(**********************************************Mesure debit ByPass*)
(*******Convertion de la pression en débit**********)
Calcul_5 := EXPT(Tab_MES_Sonde_Press_ByPass.R_MesCor,2);
Calcul_6 := EXPT(Tab_MES_Sonde_Press_ByPass.R_MesCor,1);
MES_Debit_ByPass_m3h :=  (0.0035 * Calcul_5) + (0.8986 * Calcul_6) + 10.289;

(*******Mise à zéro de la mesure en cas d'arrête*********)
TON_P1(IN:= (TON_F6.Q OR NOT Option_Mot_ByPass), PT:= T#2s);
IF (TON_P1.Q)
	THEN
	MES_Debit_ByPass_m3h := 0.0;
	ELSE
	MES_Debit_ByPass_m3h := MES_Debit_ByPass_m3h;
END_IF;

(**********************************************Mesure debit extraction et soufflage en Vol/h*)
Filtre_V1_Extraction(Mesure:= Tab_MES_Sonde_Gros_Debit_Extraction.R_MesCor, Temps_Echantillonage:= T#2s);
Filtre_V1_Soufflage(Mesure:= Tab_MES_Sonde_Gros_Debit_Soufflage.R_MesCor, Temps_Echantillonage:= T#2s);
Filtre_V1_BasDebit(Mesure:= MES_Petit_Debit_m3h_Extraction, Temps_Echantillonage:= T#1s);
Filtre_V1_ByPass(Mesure:= MES_Debit_ByPass_m3h, Temps_Echantillonage:= T#1s);

IF (Enable_PID_Bas_Deb_Ext)
	THEN
	MES_Debit_Volh_Soufflage 		:= MES_Petit_Debit_m3h_Extraction / MAX(1,Volume_Cabine);
ELSE
	MES_Debit_Volh_Soufflage			:= Filtre_V1_Soufflage.Mesure_Echantillonner / MAX(1,Volume_Cabine);
END_IF;
MES_Debit_Volh_Extraction 		:= Filtre_V1_Extraction.Mesure_Echantillonner / MAX(1,Volume_Cabine);
MES_Petit_Debit_Volh_Extraction 	:= MES_Petit_Debit_m3h_Extraction / MAX(1,Volume_Cabine);
MES_Debit_ByPass_Volh 			:= Filtre_V1_ByPass.Mesure_Echantillonner / MAX(1,Volume_Cabine);

(**********************************************Mesure de la temperature d'ambiance en °F*)
MES_Sonde_Temp_Amb_F := LIMIT(0.0, ((Tab_MES_Sonde_Temp_Amb.R_MesCor * 1.8) + 32), 100.0);

(**********************************************Mesure de la temperature de l'eau mitige de l'arrivée d'eau en °C et °F*)
IF(Option_Sonde_Temp_EauMitig) (*Option gestion régulation température eau mitigée*)
	THEN
	MES_Temp_Eau_Mitige_Cabine := Tab_MES_Sonde_Temp_Eau_Mitig.R_MesCor;
	MES_Temp_Eau_Mitige_Cabine_F := (MES_Temp_Eau_Mitige_Cabine * 1.8) + 32;
	ELSE
	MES_Temp_Eau_Mitige_Cabine := 0.0;
	MES_Temp_Eau_Mitige_Cabine_F := 0.0;
END_IF;

(**********************************************Mesure de la temperature de l'eau mitige de l'arrivée d'eau en °C et °F*)
IF(Option_Vanne_Thermo_General) (*Option vanne thermostatique présente pour toute les cabines*)
	THEN
	MES_Temp_Eau_Mitige_General_F := INT_TO_REAL(Temp_Eau_Mitige) / 10.0;
	MES_Temp_Eau_Mitige_General := LIMIT(0.0, ((MES_Temp_Eau_Mitige_General_F - 32.0) / 1.8), 100.0);
	ELSE
	MES_Temp_Eau_Mitige_General_F := 0.0;
	//MES_Temp_Eau_Mitige_General := 0.0;
END_IF;

(**********************************************Mesure sonde de pression de soufflage general*)
IF(Option_Press_SoufExt_General) (*Gestion des options*)
	THEN	E_Sonde_press_Souf := E_Sonde_press_Souf;
	ELSE	E_Sonde_press_Souf := 0;
END_IF;

(*Objet sonde*)
Objet_Sonde_V1_Press_Souf(
	Mesure_EAN:= INT_TO_REAL(E_Sonde_press_Souf),
	Enable_Alarme:= TRUE,
	Status_DEF_EAN:= FALSE,
	Tempo_AL:= T#60s,
	Hyst_AL:= 1.0,
	EAN_MIN:= 0.0,
	EAN_MAX:= 32767.0,
	MES_MIN:= 0.0,
	MES_MAX:= 500.0,
	Filtre_Actif:= TRUE,
	Temps_Echantillonage:= T#500ms,
	Tab_Sonde:= Tab_Mes_Sonde_Pression_Souf);
Tab_Mes_Sonde_Pression_Souf.R_MesCor := Tab_Mes_Sonde_Pression_Souf.R_MesCor;

(**********************************************Mesure sonde de pression d'extraction general*)
IF(Option_Press_SoufExt_General) (*Gestion des options*)
	THEN	E_Sonde_press_Ext := E_Sonde_press_Ext;
	ELSE	E_Sonde_press_Ext := 0;
END_IF;

(*Objet sonde*)
Objet_Sonde_V1_Press_Ext(
	Mesure_EAN:= INT_TO_REAL(E_Sonde_press_Ext),
	Enable_Alarme:= TRUE,
	Status_DEF_EAN:= FALSE,
	Tempo_AL:= T#60s,
	Hyst_AL:= 1.0,
	EAN_MIN:= 0.0,
	EAN_MAX:= 32767.0,
	MES_MIN:= 0.0,
	MES_MAX:= 500.0,
	Filtre_Actif:= TRUE,
	Temps_Echantillonage:= T#500ms,
	Tab_Sonde:= Tab_Mes_Sonde_Pression_Ext);
Tab_Mes_Sonde_Pression_Ext.R_MesCor := Tab_Mes_Sonde_Pression_Ext.R_MesCor;

(*********************************************Mesure sonde de température batterie eau glacée*)
IF(Option_Temp_Batterie_EG) (*Gestion des options*)
	THEN	E_Sonde_Temp_Batt_EG := E_Sonde_Temp_Batt_EG;
	ELSE	E_Sonde_Temp_Batt_EG := 0;
END_IF;

(*Objet sonde*)
Objet_Sonde_Temp_Batt_EG(
	Mesure_EAN:= INT_TO_REAL(E_Sonde_Temp_Batt_EG),
	Enable_Alarme:= FALSE,
	Status_DEF_EAN:= FALSE,
	Tempo_AL:= T#60s,
	Hyst_AL:= 1.0,
	EAN_MIN:= 0.0,
	EAN_MAX:= 32767.0,
	MES_MIN:= -15.0,
	MES_MAX:= 35.0,
	Filtre_Actif:= FALSE,
	Temps_Echantillonage:= T#1s,
	Tab_Sonde:= Tab_Mes_Sonde_Temp_BatEG);
Tab_Mes_Sonde_Temp_BatEG.R_MesCor := Tab_Mes_Sonde_Temp_BatEG.R_MesCor;

(*********************************************Mesure sonde de température au soufflage*)
IF(TRUE) (*Gestion des options*)
	THEN	E_Sonde_Temp_Souf := E_Sonde_Temp_Souf;
	ELSE	E_Sonde_Temp_Souf := 0;
END_IF;

(*Objet sonde*)
Objet_Sonde_Temp_Souf(
	Mesure_EAN:= INT_TO_REAL(E_Sonde_Temp_Souf),
	Enable_Alarme:= TRUE,
	Status_DEF_EAN:= Defaut_Sonde_Temp_Souf,
	Tempo_AL:= T#5S,
	Hyst_AL:= 1.0,
	EAN_MIN:= 0.0,
	EAN_MAX:= 32767.0,
	MES_MIN:= -20.0,
	MES_MAX:= 80.0,
	Filtre_Actif:= FALSE,
	Temps_Echantillonage:= T#1s,
	Tab_Sonde:= Tab_Mes_Sonde_Temp_Souf);
Tab_Mes_Sonde_Temp_Souf.R_MesCor := Tab_Mes_Sonde_Temp_Souf.R_MesCor;

END_PROGRAM

// ---- POUs/Block/Objets/Objet_Sonde_V1.TcPOU
FUNCTION_BLOCK Objet_Sonde_V1
VAR_INPUT
	Mesure_EAN: REAL;
	Enable_Alarme: BOOL;
	Status_DEF_EAN: BOOL;
	Tempo_AL: TIME;
	Hyst_AL: REAL;
	EAN_MIN: REAL;
	EAN_MAX: REAL;
	MES_MIN: REAL;
	MES_MAX: REAL;
	Filtre_Actif: BOOL;
	Temps_Echantillonage: TIME;
END_VAR

VAR
	TON_AL_S: TON;
	TON_AL_B: TON;
	TON_AL_H: TON;
	TON_1: TON;
	TON_2: TON;
	TP_1: TP;
	TP_2: TP;
	R_TRIG_1: R_TRIG;
	R_TRIG_2: R_TRIG;
	val_a: REAL;
	val_b: REAL;
	val_y: REAL;
	val_x: REAL;
	val_1: REAL;
	val_2: REAL;
	Diff_Mesure: REAL;
	Mesure_Echantillonner: REAL;
	Incremment_Mesure: REAL;
	Incremment_Temps: TIME;
	DINT_Temps_Echantillonage: DINT;
	DINT_Incremment_Temps: DINT;
END_VAR
VAR_IN_OUT
	Tab_Sonde :Objet_Sonde;
END_VAR

(* Gestion mesure **************************************************************)
(* Mise à l'échelle température *)
val_1 := MES_MAX - MES_MIN;
val_2 := EAN_MAX - EAN_MIN;
val_x := Mesure_EAN;
val_a := val_1 / MAX(0.1,val_2);
val_b := MES_MAX - (val_a * EAN_MAX);
val_y := (val_a * val_x) + val_b;
Tab_Sonde.R_MesBrut := LIMIT(MES_MIN,val_y,MES_MAX);

(* Gestion filtrage mesure *)
(* Fonction échantillonnage ***************)
TON_1(IN := NOT(TP_1.Q), PT := Temps_Echantillonage);
TP_1(IN := TON_1.Q , PT := T#500ms);

(* Calcule de l'éccart entre la mesure et mesure T-1 ***************) 
R_TRIG_1(CLK := TP_1.Q);
IF R_TRIG_1.Q
	THEN
		Diff_Mesure := Tab_Sonde.R_MesBrut - Mesure_Echantillonner;
END_IF;

(* Détermination de l'incremment ***************)
Incremment_Mesure := Diff_Mesure / 10.0;

(* Détermination du temps entre chaque incremmentation ***************) 
DINT_Temps_Echantillonage := TIME_TO_DINT(Temps_Echantillonage) / 1000;
DINT_Incremment_Temps := DINT_Temps_Echantillonage;
Incremment_Temps := DINT_TO_TIME(DINT_Incremment_Temps * 1000);

(* Echantillonage de la mesure ***************) 
(* Temporisation d'incrementation *)
TON_2(IN := NOT(TP_2.Q), PT := Incremment_Temps);
TP_2(IN := TON_2.Q , PT := T#100ms);

R_TRIG_2(CLK := TP_2.Q);
IF R_TRIG_2.Q
	THEN
		Mesure_Echantillonner := Mesure_Echantillonner + Incremment_Mesure;
END_IF;

(* Calcule mesure température corrigé *)
IF Filtre_Actif
	THEN
		Tab_Sonde.R_MesCor := Mesure_Echantillonner + Tab_Sonde.W_Offset;
	ELSE
		Tab_Sonde.R_MesCor := Tab_Sonde.R_MesBrut + Tab_Sonde.W_Offset;
END_IF;

(* Gestion alarmes *************************************************************)
(* Alarme status température *)
TON_AL_S(IN := Status_DEF_EAN, PT := Tempo_AL);
Tab_Sonde.Mot_Lecture.0 := TON_AL_S.Q;

(* Alarme température basse *)
TON_AL_B(IN := (Tab_Sonde.R_MesCor < Tab_Sonde.W_SeuilAlarmeBasse) AND Enable_Alarme, PT := Tempo_AL);
IF TON_AL_B.Q
	THEN
		Tab_Sonde.Mot_Lecture.2 := TRUE;
END_IF;
IF ((Tab_Sonde.R_MesCor - Hyst_AL) >= Tab_Sonde.W_SeuilAlarmeBasse OR NOT (Enable_Alarme))
	THEN
		Tab_Sonde.Mot_Lecture.2 := FALSE;
END_IF;

(* Alarme température haute *)
TON_AL_H(IN := (Tab_Sonde.R_MesCor > Tab_Sonde.W_SeuilAlarmeHaute) AND Enable_Alarme, PT := Tempo_AL);
IF TON_AL_H.Q
	THEN
		Tab_Sonde.Mot_Lecture.1 := TRUE;
END_IF;
IF ((Tab_Sonde.R_MesCor + Hyst_AL) <= Tab_Sonde.W_SeuilAlarmeHaute OR NOT (Enable_Alarme))
	THEN
		Tab_Sonde.Mot_Lecture.1 := FALSE;
END_IF;

END_FUNCTION_BLOCK

// ---- POUs/Block/Autres/Filtre_V1.TcPOU
FUNCTION_BLOCK Filtre_V1
VAR_INPUT
	Mesure: REAL;
	Temps_Echantillonage: TIME;
END_VAR
VAR_OUTPUT
	Mesure_Echantillonner: REAL;
END_VAR
VAR
	Diff_Mesure: REAL;
	Incremment_Mesure: REAL;
	Incremment_Temps: TIME;
	DINT_Temps_Echantillonage: DINT;
	DINT_Incremment_Temps: DINT;
	TON_1: TON;
	TP_1: TP;
	R_TRIG_1: R_TRIG;
	TON_2: TON;
	TP_2: TP;
	R_TRIG_2: R_TRIG;
	Temps_Ecoule: TIME;
	Temps_Incremment: TIME;
END_VAR

(* Fonction échantillonnage ***************)
TON_1(IN := NOT(TP_1.Q), PT := Temps_Echantillonage);
Temps_Ecoule := TON_1.ET;
TP_1(IN := TON_1.Q , PT := T#500ms);

(* Calcule de l'éccart entre la mesure et mesure T-1 ***************)
R_TRIG_1(CLK := TP_1.Q);
IF R_TRIG_1.Q
	THEN
		Diff_Mesure := Mesure - Mesure_Echantillonner;
END_IF;

(* Détermination de l'incremment ***************) 
Incremment_Mesure := Diff_Mesure / 10.0;

(* Détermination du temps entre chaque incremmentation ***************) 
DINT_Temps_Echantillonage := TIME_TO_DINT(Temps_Echantillonage) / 1000;
DINT_Incremment_Temps := DINT_Temps_Echantillonage;
Incremment_Temps := DINT_TO_TIME(DINT_Incremment_Temps * 1000);

(* Echantillonage de la mesure ***************) 
(* Temporisation d'incrementation *)
TON_2(IN := NOT(TP_2.Q), PT := Incremment_Temps);
Temps_Incremment := TON_2.ET;
TP_2(IN := TON_2.Q , PT := T#100ms);

R_TRIG_2(CLK := TP_2.Q);
IF R_TRIG_2.Q
	THEN
		Mesure_Echantillonner := Mesure_Echantillonner + Incremment_Mesure;
END_IF;

END_FUNCTION_BLOCK

// ---- POUs/Block/Autres/SCL.TcPOU
FUNCTION_BLOCK SCL
VAR_INPUT
	IN_INT: INT;
	LIM_MIN_IN_REAL: REAL;
	LIM_MAX_IN_REAL: REAL;
	LIM_MIN_OUT_REAL: REAL;
	LIM_MAX_OUT_REAL: REAL;
END_VAR
VAR_OUTPUT
	OUT_REAL: REAL;
	OUT_INT: INT;
END_VAR
VAR
	val_final: REAL;
	TON_1: TON;
	SCL_OUT: REAL;
	TON_2: TON;
	val_b: REAL;
	val_a: REAL;
	val_y: REAL;
	val_x: REAL;
	LIM_MAX_IN: REAL;
	LIM_MAX_OUT: REAL;
	SCL_IN: REAL;
END_VAR

(* Sécurité anti division / 0 *)

TON_1(IN := TRUE, PT := t#1s);
LIM_MAX_IN := SEL(TON_1.Q, 1.0, LIM_MAX_IN_REAL);

IF ((LIM_MAX_IN - LIM_MIN_IN_REAL) = 0.0)
	THEN
		SCL_IN := 1.0;
	ELSE
		SCL_IN := LIM_MAX_IN - LIM_MIN_IN_REAL;
END_IF;

TON_2(IN := TRUE, PT := t#1s);
LIM_MAX_OUT := SEL(TON_2.Q, 1.0, LIM_MAX_OUT_REAL);

IF ((LIM_MAX_OUT - LIM_MIN_OUT_REAL) = 0.0)
	THEN
		SCL_OUT := 1.0;
	ELSE
		SCL_OUT := LIM_MAX_OUT - LIM_MIN_OUT_REAL;
END_IF;

(* Mise à l'échelle *)

val_x := INT_TO_REAL(IN_INT);

val_b := LIM_MAX_OUT_REAL - (val_a * LIM_MAX_IN_REAL);

val_a := (SCL_OUT) / MAX(0.1,(SCL_IN));

val_y := (val_a * val_x) + val_b;


(* Traitement final *)

val_final := val_y;
OUT_REAL := LIMIT(0.0, val_final, LIM_MAX_OUT_REAL);
OUT_INT := REAL_TO_INT(OUT_REAL);

END_FUNCTION_BLOCK

// ---- POUs/c_Gestion_Defaut.TcPOU
PROGRAM c_Gestion_Defaut
VAR
(*Gestion du defaut débordement du bac à douche*)
	TON_1: TON;
	RS_Def_Debord_Douche: RS;
(*Gestion du defaut débordement du lavabo*)
	TON_2: TON;
	RS_Def_Debord_Lavabo: RS;
(*Alarme Discordance débit d'eau de douche*)
	TON_3: TON;
	RS_Deb_Eau_Douche: RS;
(*Alarme Discordance débit d'eau du lavabo*)
	TON_4: TON;
	RS_Deb_Eau_Lavabo: RS;
(*Gestion du défaut de discordance de la prise de courant*)
	TON_5: TON;
	RS_Discord_Prise: RS;
(*Gestion du défaut de discordance alimentation de la prise (si contacteur forcé manuellement)*)
	TON_6: TON;
	RS_Forcage_Prise: RS;
(*Coupure prise en cas d'ouverture de la porte lors d'une recette en cours*)
	Mode_Prise_En_Cours: BOOL;
	RS_Porte_Ouv_Cycle: RS;
(*Gestion du defaut pompe de relevage*)
	TON_7: TON;
(*Gestion du defaut ouverture de la porte trop longue*)
	TON_8: TON;
(*Gestion des défauts de communication du module dalcnet*)
	TON_ComDalcnet :TON;
	RS_Def_Com_Dalcnet: RS;
(*Gestion des défauts de communication de la vanne thermostatique otpion sur chaque cabine*)
	TON_Thermo :TON;
	RS_Def_Com_Vanne_Thermo: RS;
(*Gestion des défauts de communication de la vanne thermostatique otpion vanne general*)
	TON_ThermoGen :TON;
	RS_Def_Com_Vanne_General: RS;
(*Gestion du defaut de communication*)
	TON_Def_Client: TON;
(*Gestion du défaut discordance débit Extraction*)
	TON_9: TON;
(*Gestion du défaut discordance débit Soufflage*)
	TON_10: TON;
(*Alarme Discordance débit soufflage quand le registre Fermé*)
	TON_11: TON;
(*Alarme Discordance débit extraction quand le registre Fermé*)
	TON_12: TON;
(*Gestion du défaut différentiel de la prise électrique*)
	RS_Diff_Prise: RS;
(*Gestion des défauts de communication registre soufflage*)
	TON_ComSouf :TON;
	RS_Def_Com_Souf: RS;
(*Gestion des défauts de communication registre extraction*)
	TON_ComExt :TON;
	RS_Def_Com_Ext : RS;
(*Gestion du défaut discordance de l'ensemble bas débit*)
	TON_BasDeb :TON;
(*Gestion du défaut discordance de l'ensemble bypass*)
	TON_Bypass :TON;
(*Gestion du défaut discordance régulation de pression*)
	TON_Discord_Press: TON;
(*Gestion du défaut du capteur de pression*)
	TON_Def_Press: TON;
(*Gestion du défaut du capteur de température*)
	TON_Def_Temp: TON;
(*Gestion du défaut du capteur de hygrometrie*)
	TON_Def_Hygro: TON;
(*Gestion du défaut du capteur de température de l'eau mitigée*)
	TON_Def_Temp_Eau_Mitig: TON;
(*Gestion du défaut du capteur de température de soufflage*)
	TON_Def_Temp_Souf: TON;
END_VAR

(**********************************************Gestion du defaut débordement du bac à douche*)
IF (Option_Niveau_Haut_Douche)(*Gestion de l'option de du niveau*)
	THEN
	TON_1(IN:= (NOT E_Info_Niveau_Haut_Douche) , PT:= t#2s ); (*Temporisation en cas de coupure d'alimentation armoire*)
	RS_Def_Debord_Douche(SET:= TON_1.Q, RESET1:= Cmd_Rearmement);
	Defaut_Debordement_Douche := RS_Def_Debord_Douche.Q1;
	Defaut_Debordement_Lavabo := RS_Def_Debord_Douche.Q1;
	ELSE
	TON_1(IN:=FALSE);
	RS_Def_Debord_Douche(SET:=FALSE, RESET1:=TRUE);
	Defaut_Debordement_Douche := FALSE;
	Defaut_Debordement_Lavabo := FALSE;
END_IF;

(**********************************************Alarme Discordance débit d'eau de douche*)
IF(Option_Debitmetre_Douche)
	THEN
	TON_3(IN:= (NOT EF_Cmd_ElectroValve_Alim_Douche AND S_Cmd_ElectroValve_Alim_Douche  AND (E_Sonde_Debit_Alim_Douche <= 1000)) , PT:= t#20s );
	RS_Deb_Eau_Douche(SET:= TON_3.Q,
		RESET1:= Cmd_Rearmement,
		Q1=> Defaut_Discord_Deb_Eau_Douche);
	ELSE
	TON_3(IN:=FALSE);
	RS_Deb_Eau_Douche(SET:=FALSE, RESET1:=TRUE);
	Defaut_Discord_Deb_Eau_Douche := FALSE;
END_IF;

(**********************************************Alarme Discordance débit d'eau du lavabo*)
IF(Option_Debitmetre_Lavabo)
	THEN
	TON_4(IN:= (NOT EF_Cmd_ElectroValve_Alim_Lavabo AND S_Cmd_ElectroValve_Alim_Lavabo  AND (E_Sonde_Debit_Alim_Lavabo <= 1000)) , PT:= t#20s );
	RS_Deb_Eau_Lavabo(SET:= TON_4.Q,
		RESET1:= Cmd_Rearmement,
		Q1=> Defaut_Discord_Deb_Eau_Lavabo);
	ELSE
	TON_4(IN:=FALSE);
	RS_Deb_Eau_Lavabo(SET:=FALSE, RESET1:=TRUE);
	Defaut_Discord_Deb_Eau_Lavabo := FALSE;
END_IF;

(**********************************************Gestion du défaut de discordance de la prise de courant*)
IF(Option_Prise)
	THEN
	TON_5(IN:= (S_Cmd_PC_Cab AND NOT E_Info_PC_Cab)  , PT:= t#1s );
	RS_Discord_Prise(SET:= TON_5.Q, RESET1:= Cmd_Rearmement);
	Defaut_Discord_PC_Cab := RS_Discord_Prise.Q1;
	ELSE
	TON_5(IN:=FALSE);
	RS_Discord_Prise(SET:=FALSE, RESET1:=TRUE);
	Defaut_Discord_PC_Cab := FALSE;
END_IF;

(**********************************************Gestion du défaut de discordance alimentation de la prise (si contacteur forcé manuellement)*)
IF(Option_Prise)
	THEN
	TON_6(IN:= (NOT S_Cmd_PC_Cab AND E_Info_PC_Cab)  , PT:= t#500ms );
	RS_Forcage_Prise(SET:= (TON_6.Q), RESET1:= Cmd_Rearmement);
	Def_Discord_Alim_Prise := RS_Forcage_Prise.Q1;
	ELSE
	TON_6(IN:=FALSE);
	RS_Forcage_Prise(SET:=FALSE, RESET1:=TRUE);
	Def_Discord_Alim_Prise := FALSE;
END_IF;

(**********************************************Coupure prise en cas d'ouverture de la porte lors d'une recette en cours*)
IF(Option_Prise AND Option_Contact_Porte AND Option_Cabine_Humide AND FALSE)
	THEN
	Mode_Prise_En_Cours := Mode_Auto.Mode_6 OR Mode_Manu.Mode_6;
	RS_Porte_Ouv_Cycle(	SET:= (S_Cmd_PC_Cab AND NOT E_Info_Contact_Porte AND Mode_Prise_En_Cours),
						RESET1:= (Cmd_Rearmement OR NOT Mode_Prise_En_Cours),
						Q1 => Def_Prise_Porte_Ouverte);
	ELSE
	Mode_Prise_En_Cours := FALSE;
	RS_Porte_Ouv_Cycle(SET:=FALSE, RESET1:=TRUE);
	Def_Prise_Porte_Ouverte := FALSE;
END_IF;

(**********************************************Gestion du defaut pompe de relevage*)
IF(Option_Pompe_De_Relevage)
	THEN
	TON_7(IN:= (NOT E_Etat_Evac_SaniDouche) , PT:= t#2s ); (*Temporisation en cas de coupure d'alimentation armoire*)
	Defaut_Pompe_Relevage := TON_7.Q;
	ELSE
	TON_7(IN:=FALSE);
	Defaut_Pompe_Relevage := FALSE;
END_IF

(**********************************************Gestion du defaut ouverture de la porte trop longue*)
IF(Option_Contact_Porte)
	THEN
	TON_8(IN:= (NOT E_Info_Contact_Porte) , PT:= t#1m );
	Defaut_Porte_Ouverte := TON_8.Q;
	ELSE
	TON_8(IN:=FALSE);
	Defaut_Porte_Ouverte := FALSE;
END_IF;

(**********************************************Gestion des défauts de communication de la vanne thermostatique otpion vanne general*)
TON_ThermoGen(IN:= (Com_Ok_Vanne_Thermo) , PT:= t#2s );
IF(Option_Vanne_Thermo_General)
	THEN
	RS_Def_Com_Vanne_General(	SET:= (Error_Vanne_Thermo),
						RESET1:= (TON_ThermoGen.Q));
	Defaut_Com_Vanne_General := RS_Def_Com_Vanne_General.Q1;
	ELSE
	RS_Def_Com_Vanne_General(SET:=FALSE, RESET1:=TRUE);
	Defaut_Com_Vanne_General := FALSE;
END_IF;

(**********************************************Gestion du défaut discordance débit Extraction*)
S_Ecart_Regul_PID_Extraction := ABS(Tab_MES_Sonde_Gros_Debit_Extraction.R_MesCor - FCV_01_extraction.Cons_Pos_Dem);
TON_9(IN:= ((S_Ecart_Regul_PID_Extraction > TOL_Debit_Extraction) AND NOT Enable_PID_Bas_Deb_Ext) , PT:= t#600s );
IF(TON_9.Q AND Option_RegExt_Ultrason)
	THEN
	Defaut_Discord_Deb_Ext := TRUE;
	ELSE
	Defaut_Discord_Deb_Ext := FALSE;
END_IF;

(**********************************************Gestion du défaut discordance débit Soufflage*)
S_Ecart_Regul_PID_Soufflage := ABS(Tab_MES_Sonde_Gros_Debit_Soufflage.R_MesCor - FCV_02_soufflage.Cons_Pos_Dem);
TON_10(IN:= ((S_Ecart_Regul_PID_Soufflage > TOL_Debit_Soufflage) AND NOT Enable_PID_Bas_Deb_Ext) , PT:= t#600s );
IF(TON_10.Q AND Option_RegSouf_Ultrason)
	THEN
	Defaut_Discord_Deb_Souf := TRUE;
	ELSE
	Defaut_Discord_Deb_Souf := FALSE;
END_IF;

(**********************************************Alarme Discordance débit soufflage quand le registre Fermé*)
TON_11(IN:= ((E_Sonde_Gros_Debit_Soufflage_1 > TOL_Deb_Souf_Reg_Ferm) AND Arret_Soufflage) , PT:= t#180s);
IF(TON_11.Q)
	THEN
	Defaut_Discord_Reg_Souf_Ferm := TRUE;
	ELSE
	Defaut_Discord_Reg_Souf_Ferm := FALSE;
END_IF;

(**********************************************Alarme Discordance débit extraction quand le registre Fermé*)
TON_12(IN:= ((E_Sonde_Gros_Debit_Extraction_1 > TOL_Deb_Ext_Reg_Ferm) AND Arret_Extraction) , PT:= t#180s );
IF(TON_12.Q)
	THEN
	Defaut_Discord_Reg_Ext_Ferm := TRUE;
	ELSE
	Defaut_Discord_Reg_Ext_Ferm := FALSE;
END_IF;


(**********************************************Alarme klixon batterie électrique*)
IF(Option_Batt_Elec)
	THEN
	Defaut_Klixon_BattElec := NOT E_Info_Klixon_BattElec;
	ELSE
	Defaut_Klixon_BattElec := FALSE;
END_IF;

(***********************************************Gestion du défaut qui coupe les alimentation d'eau*)
Defaut_General_Alim_Eau := Def_Discord_Alim_Prise OR Defaut_Pompe_Relevage;

(**********************************************Gestion du défaut différentiel de la prise électrique*)
IF(Option_Prise AND Option_Defaut_Prise_Elec)
	THEN
	RS_Diff_Prise	(SET:= (E_Defaut_Prise_Elec),
				RESET1:= (Cmd_Rearmement AND NOT E_Defaut_Prise_Elec),
				Q1 => Defaut_Differentiel_Prise_Elec);
	ELSE
	RS_Diff_Prise(SET:=FALSE, RESET1:=TRUE);
	Defaut_Differentiel_Prise_Elec := FALSE;
END_IF;

(**********************************************Gestion des défauts de communication registre soufflage*)
TON_ComSouf(IN:= (Com_Ok_Reg_Souf) , PT:= t#2s );
IF(Option_Com_RegSouf_Ultrason)
	THEN
	RS_Def_Com_Souf(	SET:= (Error_Com_Reg_Souf),
						RESET1:= (TON_ComSouf.Q));
	Defaut_Com_Reg_Souf := RS_Def_Com_Souf.Q1;
	ELSE
	RS_Def_Com_Souf(SET:=FALSE, RESET1:=TRUE);
	Defaut_Com_Reg_Souf := FALSE;
END_IF;

(**********************************************Gestion des défauts de communication registre extraction*)
TON_ComExt(IN:= (Com_Ok_Reg_Extraction) , PT:= t#2s );
IF(Option_Com_RegExt_Ultrason)
	THEN
	RS_Def_Com_Ext(	SET:= (Error_RS485_Reg_Ext),
						RESET1:= (TON_ComExt.Q));
	Defaut_Com_Reg_Ext := RS_Def_Com_Ext.Q1;
	ELSE
	RS_Def_Com_Ext(SET:=FALSE, RESET1:=TRUE);
	Defaut_Com_Reg_Ext := FALSE;
END_IF;

(**********************************************Gestion du défaut discordance de l'ensemble bas débit*)
IF(Option_Bas_Debit)
	THEN
	TON_BasDeb(IN:= ((Cons_Actionneur_Moteur_BasDebit > 30.0) AND (Tab_MES_Sonde_Petit_Debit_Extraction.R_MesCor < 10.0)), PT:= T#60s, Q=> Defaut_Ensemble_Bas_Debit);
	ELSE
	Defaut_Ensemble_Bas_Debit := FALSE;
	TON_BasDeb(IN:=FALSE);
END_IF;

(**********************************************Gestion du défaut discordance de l'ensemble bypass*)
IF(Option_Mot_ByPass)
	THEN
	TON_Bypass(IN:= ((Cons_Actionneur_Moteur_ByPass > 30.0) AND (Tab_MES_Sonde_Press_ByPass.R_MesCor < 10.0)), PT:= T#60s, Q=> Defaut_Ensemble_Bypass);
	ELSE
	Defaut_Ensemble_Bypass := FALSE;
	TON_Bypass(IN:=FALSE);
END_IF;

(**********************************************Gestion du défaut discordance régulation de pression*)
TON_Discord_Press(IN:= ((S_Ecart_Regul_PID_Pression > TOL_Regul_Press) AND  Enable_PID_Press_Cab) , PT:= t#60s);
IF(TON_Discord_Press.Q)
	THEN
	Defaut_Discord_Regul_Press_Cab := TRUE;
	ELSE
	Defaut_Discord_Regul_Press_Cab := FALSE;
END_IF;

(**********************************************Gestion du défaut du capteur de pression*)
TON_Def_Press(IN:= ((-47.0 >= Tab_MES_Sonde_Press_Cab.R_MesBrut) AND  Option_Capteur_Press_Cab) , PT:= t#60s);
IF(TON_Def_Press.Q AND NOT Mode_Cabine_Automatique)
	THEN
	Defaut_Sonde_Press_Cabine := TRUE;
	ELSE
	Defaut_Sonde_Press_Cabine := FALSE;
END_IF;

(**********************************************Gestion du défaut du capteur de température ambiance*)
TON_Def_Temp(IN:= ((-17.0 >= Tab_MES_Sonde_Temp_Amb.R_MesBrut) AND ( Option_Sonde_Temp_Hygro_Amb OR Option_Sonde_Temp_Amb)) , PT:= t#60s);
IF(TON_Def_Temp.Q)
	THEN
	Defaut_Sonde_Temp_Cabine := TRUE;
	ELSE
	Defaut_Sonde_Temp_Cabine := FALSE;
END_IF;

(**********************************************Gestion du défaut du capteur de hygrométrie *)
TON_Def_Hygro(IN:= ((1.0 >= Tab_MES_Sonde_Hygro_Amb.R_MesBrut) AND ( Option_Sonde_Temp_Hygro_Amb)) , PT:= t#60s);
IF(TON_Def_Hygro.Q)
	THEN
	Defaut_Sonde_Hygro_Cabine := TRUE;
	ELSE
	Defaut_Sonde_Hygro_Cabine := FALSE;
END_IF;

(**********************************************Gestion du défaut du capteur de température de l'eau mitigée*)
TON_Def_Temp_Eau_Mitig(IN:= ((-17.0 >= Tab_MES_Sonde_Temp_Eau_Mitig.R_MesBrut) AND (Option_Sonde_Temp_EauMitig)) , PT:= t#60s);
IF(TON_Def_Temp_Eau_Mitig.Q)
	THEN
	Defaut_Sonde_Temp_Eau_Mitig := TRUE;
	ELSE
	Defaut_Sonde_Temp_Eau_Mitig := FALSE;
END_IF;

(**********************************************Gestion du défaut du capteur de température de soufflage*)
TON_Def_Temp_Souf(IN:= ((-17.0 >= Tab_Mes_Sonde_Temp_Souf.R_MesBrut)) , PT:= T#60S);
IF(TON_Def_Temp_Souf.Q)
	THEN
	Defaut_Sonde_Temp_Souf := TRUE;
	ELSE
	Defaut_Sonde_Temp_Souf := FALSE;
END_IF;

(**********************************************Gestion du mode Cabine en défaut qui fait clignoter la cabine en rouge*)
Mode_Cabine_Defaut :=(
Defaut_Debordement_Douche OR Defaut_Debordement_Lavabo OR Defaut_Discord_Deb_Eau_Douche OR Defaut_Discord_Deb_Eau_Lavabo
OR Defaut_Discord_PC_Cab OR Def_Discord_Alim_Prise OR Def_Prise_Porte_Ouverte OR Defaut_Pompe_Relevage
OR Defaut_Discord_Vanne_Vid_Douche_Ouv OR Defaut_Discord_Vanne_Vid_Douche_Ferm OR Defaut_Discord_Vanne_Vid_Lavabo_Ouv OR Defaut_Discord_Vanne_Vid_Lavabo_Ferm
OR Defaut_Discord_Vanne_Alim_Douche_Ouv OR Defaut_Discord_Vanne_Alim_Douche_Ferm OR Defaut_Discord_Vanne_Alim_Lavabo_Ouv OR Defaut_Discord_Vanne_Alim_Lavabo_Ferm
OR Defaut_Discord_Vanne_Alim_Douchette_Ouv OR Defaut_Discord_Vanne_Alim_Douchette_Ferm OR Defaut_Klixon_BattElec OR Defaut_Differentiel_Prise_Elec
OR Defaut_Discord_Vanne_Souf_Bas_Deb_Ouv OR Defaut_Discord_Vanne_Souf_Bas_Deb_Ferm OR Defaut_Discord_Vanne_Ext_Bas_Deb_Ouv OR Defaut_Discord_Vanne_Ext_Bas_Deb_Ferm
OR Defaut_Discord_Reg_Etanche_Ext OR Defaut_Discord_Reg_Etanche_Ext OR Defaut_Sonde_Press_Cabine OR Defaut_Sonde_Temp_Eau_Mitig
OR Defaut_Discord_Vanne_Alim_NEP_Ouv OR Defaut_Discord_Vanne_Alim_NEP_Ferm OR Defaut_Arret_Mode25);

END_PROGRAM

// ---- POUs/d_Gestion_Pause_Modes.TcPOU
PROGRAM d_Gestion_Pause_Modes
VAR
	R_TRIG_Pause: R_TRIG;
	RS_Commande_Pause: RS;
	RS_Statut_Pause: RS;
END_VAR

(*Gestion des alarmes de sécurité qui met en pause les recettes automatiques et manuelles*)

(**********************************************Defaut du mode 1 Douche avec vidange*)
Alarme_Secu_Mode_1 := (Mode_Auto.Mode_1 OR Mode_Manu.Mode_1)
	AND (Def_Discord_Alim_Prise OR Defaut_Pompe_Relevage OR Defaut_Com_Vanne_Thermo OR Defaut_Com_Vanne_General
	OR Defaut_Discord_Vanne_Vid_Douche_Ouv OR Defaut_Discord_Vanne_Vid_Douche_Ferm
	OR Defaut_Discord_Vanne_Alim_Douche_Ouv OR Defaut_Discord_Vanne_Alim_Douche_Ferm);

(**********************************************Defaut du mode 2 Douche sans vidange*)
Alarme_Secu_Mode_2 := (Mode_Auto.Mode_2 OR Mode_Manu.Mode_2)
	AND (Def_Discord_Alim_Prise OR Defaut_Pompe_Relevage OR Defaut_Com_Vanne_Thermo OR Defaut_Com_Vanne_General
	OR Defaut_Discord_Vanne_Alim_Douche_Ouv OR Defaut_Discord_Vanne_Alim_Douche_Ferm);

(**********************************************Defaut du mode 4 Lavabo avec vidange*)
Alarme_Secu_Mode_4 := (Mode_Auto.Mode_4 OR Mode_Manu.Mode_4)
	AND (Def_Discord_Alim_Prise OR Defaut_Pompe_Relevage OR Defaut_Com_Vanne_Thermo OR Defaut_Com_Vanne_General
	OR Defaut_Discord_Vanne_Vid_Lavabo_Ouv OR Defaut_Discord_Vanne_Vid_Lavabo_Ferm
	OR Defaut_Discord_Vanne_Alim_Lavabo_Ouv OR Defaut_Discord_Vanne_Alim_Lavabo_Ferm);

(**********************************************Defaut du mode 5 Lavabo sans vidange*)
Alarme_Secu_Mode_5 := (Mode_Auto.Mode_5 OR Mode_Manu.Mode_5)
	AND (Def_Discord_Alim_Prise OR Defaut_Pompe_Relevage OR Defaut_Com_Vanne_Thermo OR Defaut_Com_Vanne_General
	OR Defaut_Discord_Vanne_Alim_Lavabo_Ouv OR Defaut_Discord_Vanne_Alim_Lavabo_Ferm);

(**********************************************Defaut du mode 6 prise*)
Alarme_Secu_Mode_6 := (Mode_Auto.Mode_6 OR Mode_Manu.Mode_6)
	AND (Defaut_Discord_PC_Cab OR Def_Prise_Porte_Ouverte
	OR Defaut_Discord_Vanne_Alim_Douche_Ferm OR Defaut_Discord_Vanne_Alim_Lavabo_Ferm
	OR Defaut_Discord_Vanne_Alim_Douchette_Ferm OR Defaut_Differentiel_Prise_Elec);

(**********************************************Defaut du mode 7 mode vidange*)
IF(Option_Douche)					(*Type de cabine douche uniquement*)
	THEN
	Alarme_Secu_Mode_7 := (Mode_Auto.Mode_7 OR Mode_Manu.Mode_7)
	AND (Defaut_Pompe_Relevage
	OR Defaut_Discord_Vanne_Vid_Douche_Ouv OR Defaut_Discord_Vanne_Vid_Douche_Ferm);
END_IF;
IF(Option_Lavabo)						(*Type de cabine lavabo uniquement*)
	THEN
	Alarme_Secu_Mode_7 := (Mode_Auto.Mode_7 OR Mode_Manu.Mode_7)
	AND (Defaut_Pompe_Relevage
	OR Defaut_Discord_Vanne_Vid_Lavabo_Ouv OR Defaut_Discord_Vanne_Vid_Lavabo_Ferm);
END_IF;
IF(Option_Lavabo AND Option_Douche)	(*Type de cabine lavabo ET douche*)
	THEN
	Alarme_Secu_Mode_7 := (Mode_Auto.Mode_7 OR Mode_Manu.Mode_7)
	AND (Defaut_Pompe_Relevage
	OR Defaut_Discord_Vanne_Vid_Lavabo_Ouv OR Defaut_Discord_Vanne_Vid_Lavabo_Ferm
	OR Defaut_Discord_Vanne_Vid_Douche_Ouv OR Defaut_Discord_Vanne_Vid_Douche_Ferm);
END_IF;

(**********************************************Defaut du mode 18 Lavage NEP chaud*)
Alarme_Secu_Mode_18 := (Mode_Auto.Mode_18 OR Mode_Manu.Mode_18)
	AND (Defaut_Discord_Vanne_Vid_Douche_Ouv OR Defaut_Discord_Vanne_Vid_Douche_Ferm
	OR Defaut_Discord_Vanne_Alim_NEP_Ouv OR Defaut_Discord_Vanne_Alim_NEP_Ferm);

(**********************************************Defaut du mode 19 Lavage NEP chaud*)
Alarme_Secu_Mode_18 := (Mode_Auto.Mode_19 OR Mode_Manu.Mode_19)
	AND (Defaut_Discord_Vanne_Vid_Douche_Ouv OR Defaut_Discord_Vanne_Vid_Douche_Ferm
	OR Defaut_Discord_Vanne_Alim_NEP_Ouv OR Defaut_Discord_Vanne_Alim_NEP_Ferm);

(**********************************************Gestion de la pause*)
R_TRIG_Pause(CLK:= Bp_Pause);
RS_Commande_Pause(
SET:=  ((NOT RS_Commande_Pause.Q1 AND R_TRIG_Pause.Q)
					OR Alarme_Secu_Mode_1 OR Alarme_Secu_Mode_2 OR Alarme_Secu_Mode_3 OR Alarme_Secu_Mode_4 OR Alarme_Secu_Mode_5
					OR Alarme_Secu_Mode_6 OR Alarme_Secu_Mode_7 OR Alarme_Secu_Mode_8 OR Alarme_Secu_Mode_10 OR Alarme_Secu_Mode_11
					OR Alarme_Secu_Mode_12 OR Alarme_Secu_Mode_13 OR Alarme_Secu_Mode_14 OR Alarme_Secu_Mode_15 OR Alarme_Secu_Mode_16
					OR Alarme_Secu_Mode_17 OR Alarme_Secu_Mode_18 OR Alarme_Secu_Mode_19 OR Alarme_Secu_Mode_23 OR Alarme_Secu_Mode_24),
RESET1:= ((RS_Commande_Pause.Q1 AND R_TRIG_Pause.Q)
					AND  (NOT Alarme_Secu_Mode_1 AND NOT Alarme_Secu_Mode_2 AND NOT Alarme_Secu_Mode_3 AND NOT Alarme_Secu_Mode_4 AND NOT Alarme_Secu_Mode_5
					AND NOT Alarme_Secu_Mode_6 AND NOT Alarme_Secu_Mode_7 AND NOT Alarme_Secu_Mode_8 AND NOT Alarme_Secu_Mode_10 AND NOT Alarme_Secu_Mode_11
					AND NOT Alarme_Secu_Mode_12 AND NOT Alarme_Secu_Mode_13 AND NOT Alarme_Secu_Mode_14 AND NOT Alarme_Secu_Mode_15 AND NOT Alarme_Secu_Mode_16
					 AND NOT Alarme_Secu_Mode_17 AND NOT Alarme_Secu_Mode_18 AND NOT Alarme_Secu_Mode_19 AND NOT Alarme_Secu_Mode_23 AND NOT Alarme_Secu_Mode_24))
					OR (NOT Mode_Cabine_Automatique AND NOT Mode_Cabine_Manuel),
Q1=> Comande_Pause);

(**********************************************Gestion de la commande pause. Seulement pour affichage IHM*)
RS_Statut_Pause(
SET:=(Alarme_Secu_Mode_1 OR Alarme_Secu_Mode_2 OR Alarme_Secu_Mode_3 OR Alarme_Secu_Mode_4 OR Alarme_Secu_Mode_5
					OR Alarme_Secu_Mode_6 OR Alarme_Secu_Mode_7 OR Alarme_Secu_Mode_8 OR Alarme_Secu_Mode_10 OR Alarme_Secu_Mode_11
					OR Alarme_Secu_Mode_12 OR Alarme_Secu_Mode_13 OR Alarme_Secu_Mode_14 OR Alarme_Secu_Mode_15 OR Alarme_Secu_Mode_16
					OR Alarme_Secu_Mode_17 OR Alarme_Secu_Mode_18 OR Alarme_Secu_Mode_19 OR Alarme_Secu_Mode_23 OR Alarme_Secu_Mode_24),
RESET1:= Bp_Pause AND (NOT Alarme_Secu_Mode_1 OR NOT Alarme_Secu_Mode_2 OR NOT Alarme_Secu_Mode_3 OR NOT Alarme_Secu_Mode_4 OR NOT Alarme_Secu_Mode_5
					OR NOT Alarme_Secu_Mode_6 OR NOT Alarme_Secu_Mode_7 OR NOT Alarme_Secu_Mode_8 OR NOT Alarme_Secu_Mode_10 OR NOT Alarme_Secu_Mode_11
					OR NOT Alarme_Secu_Mode_12 OR NOT Alarme_Secu_Mode_13 OR NOT Alarme_Secu_Mode_14 OR NOT Alarme_Secu_Mode_15 OR NOT Alarme_Secu_Mode_16
					 OR NOT Alarme_Secu_Mode_17 OR NOT Alarme_Secu_Mode_18 OR NOT Alarme_Secu_Mode_19 OR NOT Alarme_Secu_Mode_23 OR NOT Alarme_Secu_Mode_24)
					OR (NOT Mode_Cabine_Automatique AND NOT Mode_Cabine_Manuel),
Q1=> Statut_Pause_Force);

Attente_Reset_Pause := (Alarme_Secu_Mode_1 OR Alarme_Secu_Mode_2 OR Alarme_Secu_Mode_3 OR Alarme_Secu_Mode_4 OR Alarme_Secu_Mode_5
					OR Alarme_Secu_Mode_6 OR Alarme_Secu_Mode_7 OR Alarme_Secu_Mode_8 OR Alarme_Secu_Mode_10 OR Alarme_Secu_Mode_11
					OR Alarme_Secu_Mode_12 OR Alarme_Secu_Mode_13 OR Alarme_Secu_Mode_14 OR Alarme_Secu_Mode_15 OR Alarme_Secu_Mode_16
					OR Alarme_Secu_Mode_17 OR Alarme_Secu_Mode_18 OR Alarme_Secu_Mode_19 OR Alarme_Secu_Mode_23 OR Alarme_Secu_Mode_24);

END_PROGRAM

// ---- POUs/e_Gestion_Horraire.TcPOU
PROGRAM e_Gestion_Horraire
VAR
	bFirstTime	: BOOL;
	Forc_MAL: BOOL := TRUE;
	DayOfWeek: WORD;

	fbRtc		: RTC_EX2;
	fbGetTime	: NT_GetTime;
	fbSetTime	: NT_SetLocalTime;

	F_TRIG_MAL: F_TRIG;
	TOF_For_MAL: TOF;
	RTC_Time_Lum:RTC_Time;
	TOF_Occup: TOF;
	Out_Schedule: BOOL;
END_VAR

(*Variables mise à l'heure de la CPU*)
RTC_Modifiable.wYear := Ecr_Annee_Automate;
RTC_Modifiable.wMonth := Ecr_Mois_Automate;
RTC_Modifiable.wDay := Ecr_Jour_Automate;
RTC_Modifiable.wHour := Ecr_Heure_Automate;
RTC_Modifiable.wMinute := Ecr_Minute_Automate;
(*Récupération du jour de la semaine*)
DayOfWeek := F_GetDayOfWeek(SYSTEMTIME_TO_DT(RTC_Modifiable));
RTC_Modifiable.wDayOfWeek := DayOfWeek;

(*Mise à l'heure de la CPU*)
fbSetTime(
	TIMESTR	:= RTC_Modifiable,
	START		:= StartMiseALheure,
	TMOUT		:= DEFAULT_ADS_TIMEOUT);
(*Mise à l'heure de l'automate après l'ecriture de la modification de l'heure*)
F_TRIG_MAL(CLK:= StartMiseALheure, Q=> bFirstTime);

(*Récupération de l'heure depuis la CPU*)
fbGetTime(
	START		:= bFirstTime OR TOF_For_MAL.Q ,
	TMOUT		:= DEFAULT_ADS_TIMEOUT);

IF NOT fbGetTime.BUSY AND NOT fbGetTime.ERR THEN
	rtcTime := fbGetTime.TIMESTR;
	bFirstTime := FALSE;
END_IF;

(******************************RTC Time******************************)
fbRtc(
	EN 		:= NOT bFirstTime AND NOT TOF_For_MAL.Q,
	PDT 	:=rtcTime ,
	PMICRO	:= rtcMicro,
	CDT	=> rtcTime,
	CMICRO	=> rtcMicro);
(*Fonction démarrage mise à l'heure automatiquement après une mise en RUN de l'automate*)
TOF_For_MAL(IN:= Forc_MAL, PT:= T#1s);
IF (TOF_For_MAL.Q) THEN Forc_MAL := FALSE; END_IF;

(******************************Récupération Heure,Minutes,Secondes******************************)
Van := fbRtc.CDT.wYear;
Vmois :=fbRtc.CDT.wMonth;
Vjour := fbRtc.CDT.wDay;
Vheure := fbRtc.CDT.wHour;
Vminute := fbRtc.CDT.wMinute;
Vseconde := fbRtc.CDT.wSecond;
VDayOfWeek := fbRtc.CDT.wDayOfWeek;

(******************************Gestion de l'horodatage******************************)
RTC_Time_Lum(
	Auto_manu:= TRUE,
	IN_MONTH:= Vmois,
	IN_DAY:= Vjour,
	IN_HOURS:= Vheure,
	IN_MINUTES:= Vminute,
	pos_sem:= DayOfWeek,
	Heure_debut_lun:= deb_lundi,
	Heure_fin_lun:= Fin_Lundi,
	Heure_debut_mar:= deb_Mardi,
	Heure_fin_mar:= Fin_Mardi,
	Heure_debut_mer:= deb_Mercredi,
	Heure_fin_mer:= Fin_Mercredi,
	Heure_debut_jeu:= deb_Jeudi,
	Heure_fin_jeu:= Fin_Jeudi,
	Heure_debut_ven:= deb_Vendredi,
	Heure_fin_ven:= Fin_Vendredi,
	Heure_debut_sam:= deb_Samedi,
	Heure_fin_sam:= Fin_Samedi,
	Heure_debut_dim:= deb_Dimanche,
	Heure_fin_dim:= Fin_Dimanche,
	fct_hebdo:= TRUE,
	hebdo_lun:= Sel_Lundi,
	hebdo_mar:= Sel_Mardi,
	hebdo_mer:= Sel_Mercredi,
	hebdo_jeu:= Sel_Jeudi,
	hebdo_ven:= Sel_Vendredi,
	hebdo_sam:= Sel_Samedi,
	hebdo_dim:= Sel_Dimanche,
	Sortie=> Out_Schedule);
(*Temporisation en cas de paramétrage de l'heure deb 00h00 et fin 23h59*)
TOF_Occup(IN:= Out_Schedule, PT:= T#125s);
Mode_Occupation := TOF_Occup.Q;

END_PROGRAM

// ---- POUs/Block/Autres/RTC_Time.TcPOU
(*Version 1.0		Date 20.12.01*)
FUNCTION_BLOCK RTC_Time
VAR
	Jours_Mois_courant		: INT;	(* Jour courant API 3112 *)
	Heure_Minute_courant		: INT;	(* Heure courant API 2359 *)
END_VAR
VAR_INPUT
	Auto_manu				: BOOL;	(*Selection mode Auto=1/manu=0  *)
	F_On					: BOOL;	(* Forcage en mode manu ON *)
	IN_MONTH				: WORD;
	IN_DAY					: WORD;
	IN_HOURS				: WORD;	(* System TIME (hours) *)
	IN_MINUTES				: WORD;	(*System TIME (minutes)  *)
	pos_sem				: WORD;	(* Jour de la semaine*)
	Heure_debut_lun			: INT;	(* Heure de début 2359 *)
	Heure_fin_lun				: INT;	(* Heure de fin 2359 *)
	Heure_debut_mar			: INT;	(*Heure de début 2359  *)
	Heure_fin_mar			: INT;	(*Heure de fin 2359  *)
	Heure_debut_mer			: INT;	(* Heure de début 2359 *)
	Heure_fin_mer			: INT;	(* Heure de fin 2359 *)
	Heure_debut_jeu			: INT;	(* Heure de début 2359 *)
	Heure_fin_jeu				: INT;	(* Heure de fin 2359 *)
	Heure_debut_ven			: INT;	(* Heure de début 2359 *)
	Heure_fin_ven			: INT;	(* Heure de fin 2359 *)
	Heure_debut_sam			: INT;	(* Heure de début 2359 *)
	Heure_fin_sam			: INT;	(* Heure de fin 2359 *)
	Heure_debut_dim			: INT;	(* Heure de début 2359 *)
	Heure_fin_dim			: INT;	(* Heure de fin 2359 *)
	fct_periode				: BOOL;	(* Fonction Periode entre 2 dates *)
	Jour_debut				: INT;	(* Jour de début 3112 *)
	Jour_fin					: INT;	(* Jour de fin 3112 *)
	fct_hebdo				: BOOL;	(*  *)
	hebdo_lun				: BOOL;	(*  *)
	hebdo_mar				: BOOL;	(*  *)
	hebdo_mer				: BOOL;	(*  *)
	hebdo_jeu				: BOOL;	(*  *)
	hebdo_ven				: BOOL;	(*  *)
	hebdo_sam				: BOOL;	(*  *)
	hebdo_dim				: BOOL;	(*  *)
END_VAR
VAR_OUTPUT
	Sortie					: BOOL;	(*Commande de la sortie  *)
	Marche_periode			: BOOL;	(*Status état dans la periode  *)
	Marche_horaire_lun		: BOOL;	(*Status état dans la tranche horaire  *)
	Marche_horaire_mar		: BOOL;	(*Status état dans la tranche horaire *)
	Marche_horaire_mer		: BOOL;	(*Status état dans la tranche horaire  *)
	Marche_horaire_jeu		: BOOL;	(*Status état dans la tranche horaire  *)
	Marche_horaire_ven		: BOOL;	(*Status état dans la tranche horaire  *)
	Marche_horaire_sam		: BOOL;	(*Status état dans la tranche horaire  *)
	Marche_horaire_dim		: BOOL;	(*Status état dans la tranche horaire  *)
	Marche_hebdo			: BOOL;	(*  *)
	Marche_hebdo_lun		: BOOL;	(*  *)
	Marche_hebdo_mar		: BOOL;	(*  *)
	Marche_hebdo_mer		: BOOL;	(*  *)
	Marche_hebdo_jeu		: BOOL;	(*  *)
	Marche_hebdo_ven		: BOOL;	(*  *)
	Marche_hebdo_sam		: BOOL;(*  *)
	Marche_hebdo_dim		: BOOL;	(*  *)
END_VAR
VAR_EXTERNAL

END_VAR

(*Reprise infORmation système*)
Heure_Minute_courant 	:= UINT_TO_INT((IN_HOURS * 100) + IN_MINUTES);
Jours_Mois_courant 		:= UINT_TO_INT((IN_DAY * 100) + IN_MONTH);

(*LUNDI*)
IF (Heure_debut_lun < Heure_fin_lun)
	THEN
	(*fonctionnement horaire*)
		IF ( Heure_debut_lun < Heure_Minute_courant AND Heure_Minute_courant < Heure_fin_lun AND pos_sem = 1)
			THEN
				Marche_horaire_lun := TRUE;
			ELSE
				Marche_horaire_lun := FALSE;
		END_IF;
	ELSE
	Marche_horaire_lun := FALSE;
END_IF;

(*MARDI*)
IF (Heure_debut_mar < Heure_fin_mar) 
	THEN
	(*fonctionnement horaire*)
		IF ( Heure_debut_mar < Heure_Minute_courant AND Heure_Minute_courant < Heure_fin_mar AND pos_sem = 2) 
			THEN
				Marche_horaire_mar := TRUE;
			ELSE
				Marche_horaire_mar := FALSE;
		END_IF;
	ELSE
	Marche_horaire_mar := FALSE;
END_IF;

(*MERCREDI*)
IF (Heure_debut_mer < Heure_fin_mer) 
	THEN
	(*fonctionnement horaire*)
		IF ( Heure_debut_mer < Heure_Minute_courant AND Heure_Minute_courant < Heure_fin_mer AND pos_sem = 3) 
			THEN
				Marche_horaire_mer := TRUE;
			ELSE
				Marche_horaire_mer := FALSE;
		END_IF;
	ELSE
	Marche_horaire_mer := FALSE;
END_IF;

(*JEUDI*)
IF (Heure_debut_jeu < Heure_fin_jeu) 
	THEN
	(*fonctionnement horaire*)
		IF ( Heure_debut_jeu < Heure_Minute_courant AND Heure_Minute_courant < Heure_fin_jeu AND pos_sem = 4) 
			THEN
				Marche_horaire_jeu := TRUE;
			ELSE
				Marche_horaire_jeu := FALSE;
		END_IF;
	ELSE
	Marche_horaire_jeu := FALSE;
END_IF;

(*VENDREDI*)
IF (Heure_debut_ven < Heure_fin_ven) 
	THEN
	(*fonctionnement horaire*)
		IF ( (Heure_debut_ven < Heure_Minute_courant) AND( Heure_Minute_courant < Heure_fin_ven) AND (pos_sem = 5))
			THEN
				Marche_horaire_ven := TRUE;
			ELSE
				Marche_horaire_ven := FALSE;
		END_IF;
	ELSE
	Marche_horaire_ven := FALSE;
END_IF;

(*SAMEDI*)
IF (Heure_debut_sam < Heure_fin_sam) 
	THEN
	(*fonctionnement horaire*)
		IF ( Heure_debut_sam < Heure_Minute_courant AND Heure_Minute_courant < Heure_fin_sam AND pos_sem = 6) 
			THEN
				Marche_horaire_sam := TRUE;
			ELSE
				Marche_horaire_sam := FALSE;
		END_IF;
	ELSE
	Marche_horaire_sam := FALSE;
END_IF;

(*DIMANCHE*)
IF (Heure_debut_dim < Heure_fin_dim)
	THEN
	(*fonctionnement horaire*)
		IF ( Heure_debut_dim < Heure_Minute_courant AND Heure_Minute_courant < Heure_fin_dim AND pos_sem = 0) 
			THEN
				Marche_horaire_dim := TRUE;
			ELSE
				Marche_horaire_dim := FALSE;
		END_IF;
	ELSE
	Marche_horaire_dim := FALSE;
END_IF;

(*Fonctionnement periodique*)
Marche_periode := FALSE;
IF ( fct_periode = TRUE ) 
	THEN
		IF ( Jour_debut <= Jour_fin) 
			THEN
				IF ( Jour_debut <= Jours_Mois_courant AND Jours_Mois_courant <= Jour_fin ) 
					THEN
						Marche_periode := TRUE;
					ELSE
						Marche_periode := FALSE;
				END_IF;
			ELSE
			(*Fonctionnement a cheval sur 2 année*)
				IF ( Jour_debut <= Jours_Mois_courant AND Jours_Mois_courant <= Jour_fin ) 
					THEN
						Marche_periode := FALSE;
					ELSE
						Marche_periode := TRUE;
				END_IF;
		END_IF;
	ELSE
		Marche_periode:=TRUE;
END_IF;

(*Fonctionnement hebdomatdaire*)
Marche_hebdo := FALSE;
Marche_hebdo_lun := FALSE;
Marche_hebdo_mar := FALSE;
Marche_hebdo_mer := FALSE;
Marche_hebdo_jeu := FALSE;
Marche_hebdo_ven := FALSE;
Marche_hebdo_sam := FALSE;
Marche_hebdo_dim := FALSE;

IF ( fct_hebdo = TRUE )
	THEN
		IF ( hebdo_lun = TRUE AND pos_sem = 1)
			THEN
				Marche_hebdo_lun := TRUE;	
		END_IF;
		IF ( hebdo_mar = TRUE AND pos_sem = 2) 
			THEN
				Marche_hebdo_mar := TRUE;
		END_IF;
		IF ( hebdo_mer = TRUE AND pos_sem = 3) 
			THEN
				Marche_hebdo_mer := TRUE;
			END_IF;
		IF ( hebdo_jeu = TRUE AND pos_sem = 4) 
			THEN
				Marche_hebdo_jeu := TRUE;
		END_IF;
		IF ( hebdo_ven = TRUE AND pos_sem = 5) 
			THEN
				Marche_hebdo_ven := TRUE;
			END_IF;
		IF ( hebdo_sam = TRUE AND pos_sem = 6) 
			THEN
				Marche_hebdo_sam := TRUE;
			END_IF;
		IF ( hebdo_dim = TRUE AND pos_sem = 7)
			THEN
				Marche_hebdo_dim := TRUE;
			END_IF;
	ELSE
		Marche_hebdo := TRUE;
END_IF;

(*Gestion Auto/manu et On/Off*)
Sortie := FALSE;
IF (Auto_manu = TRUE) 
	THEN
	(*Selection horaire*)
		IF (Marche_periode = TRUE 
			AND (
				(Marche_hebdo_lun = TRUE AND Marche_horaire_lun = TRUE) 
				OR (Marche_hebdo_mar = TRUE AND Marche_horaire_mar = TRUE) 
				OR (Marche_hebdo_mer = TRUE AND Marche_horaire_mer = TRUE) 
				OR (Marche_hebdo_jeu = TRUE AND Marche_horaire_jeu = TRUE) 
				OR (Marche_hebdo_ven = TRUE AND Marche_horaire_ven = TRUE) 
				OR (Marche_hebdo_sam = TRUE AND Marche_horaire_sam = TRUE) 
				OR (Marche_hebdo_dim = TRUE AND Marche_horaire_dim = TRUE)
				)
			) 
			THEN
				Sortie := TRUE;
		END_IF;
	ELSE
		IF ( F_On = TRUE ) 
			THEN
				Sortie := TRUE;
		ELSE
			Sortie := FALSE;
		END_IF;
END_IF;

END_FUNCTION_BLOCK

// ---- POUs/f_Gestion_Etats.TcPOU
PROGRAM f_Gestion_Etats
VAR
(*Gestion etat cabine dépollution*)
	RS_Depollution: RS;
	R_TRIG_Depol: R_TRIG;
	TON_Depollution: TON_V1;
	R_TRIG_cylcle1: R_TRIG;
	TP_Cycle1: TP;
	RS_CTA: RS;
(*Gestion etat cabine Manuel*)
	Mode_END_Manu: BOOL;
	Securite_Tempo_Manu: REAL;
	RS_Manu: RS;
(*Gestion etat cabine Automatique*)
	Mode_END_Auto: BOOL;
	RS_Automatique: RS;
(*Gestion de la condition d'affichage du bouton étape suivante*)
	Mode_texte_Auto: BOOL;
	Mode_Evaluation_Auto: BOOL;
	Mode_Netoyage_Auto: BOOL;
	Mode_Lav_Douch_Bouton_Auto: BOOL;
	Mode_MiseEnCondi: BOOL;
	R_TRIG_FIN: R_TRIG;
END_VAR

(**********************************************Gestion de la condition d'affichage du bouton étape suivante*)
(*Affichage du bouton étape suivante si mode 30 à 59 OU mode 24 OU mode 23 OU mode 3 OU mode 16 OU mode 17 *)
Mode_texte_Auto				:= (Mode_Auto.Numero_Mode >= 30) AND (Mode_Auto.Numero_Mode <= 59);
Mode_Evaluation_Auto		:= Mode_Auto.Mode_23 OR Mode_Auto.Mode_24;
Mode_Netoyage_Auto			:= Mode_Auto.Mode_3;
Mode_Lav_Douch_Bouton_Auto	:= Mode_Auto.Mode_16 OR Mode_Auto.Mode_17;
Mode_MiseEnCondi			:= Mode_Auto.Mode_25 OR Mode_Auto.Mode_28;
IF (Mode_texte_Auto OR Mode_Evaluation_Auto OR Mode_Netoyage_Auto OR Mode_Lav_Douch_Bouton_Auto OR Mode_MiseEnCondi)
	THEN
	Condi_Affich_Etape_Suiv := TRUE;
	ELSE
	Condi_Affich_Etape_Suiv := FALSE;
END_IF;


(********************************************** Gestion de l'affichage du bouton de réarmement*)
IF (Defaut_Debordement_Douche OR Defaut_Debordement_Lavabo OR Defaut_Discord_Deb_Eau_Douche OR Defaut_Discord_Deb_Eau_Lavabo
	OR Defaut_Discord_PC_Cab OR Def_Discord_Alim_Prise OR Def_Prise_Porte_Ouverte OR Defaut_Differentiel_Prise_Elec OR Defaut_Thermostat_Secu)
	THEN
	Condi_Affich_Rearm := TRUE;
	ELSE
	Condi_Affich_Rearm := FALSE;
END_IF;

(************************************************Gestion du mode Neutre et Evaluation*)
Mode_Evaluation := Mode_Auto.Mode_23 OR Mode_Auto.Mode_24;
Mode_Neutre := Mode_Auto.Mode_8 OR Mode_Manu.Mode_8;

(*************************************************Gestion de la commande de la régulation de l'extraction*)
IF((Mode_Neutre  OR (Cons_Actionneur_Registre_Ext_Volh = 0)))
	THEN
	Arret_Extraction := TRUE;
	ELSE
	Arret_Extraction := FALSE;
END_IF;

(*************************************************Gestion de la commande de la régulation du soufflage*)
IF((Mode_Neutre OR (Cons_Actionneur_Registre_Souf_Volh = 0)))
	THEN
	Arret_Soufflage := TRUE;
	ELSE
	Arret_Soufflage := FALSE;
END_IF;

(**************************************************Gestion etat cabine éclairage*)
IF(Activation_Ecl)
	THEN
	Mode_Cabine_Eclairage := TRUE;
	ELSE
	Mode_Cabine_Eclairage := FALSE;
END_IF;

(***************************************************Gestion etat cabine dépollution*)
R_TRIG_Depol(CLK:= Start_Etat_Depollution);
RS_Depollution(
SET:= (R_TRIG_Depol.Q AND NOT RS_Depollution.Q1),
RESET1:= 	(Mode_Cabine_Automatique OR Mode_Cabine_Manuel OR Mode_Maintenance)
			OR (R_TRIG_Depol.Q AND RS_Depollution.Q1) OR TON_Depollution.Q);

TON_Depollution(
	Enable:= RS_Depollution.Q1,
	Pause:= ,
	In_Cons_Seconde:= 1,
	In_Cons_Minute:= Cons_Temp_Minute_Depol,
	In_Cons_Heure:= Cons_Temp_heure_Depol,
	In_Cons_Jour:= 0 ,
	Seconde_Restant=> Lect_Temp_Seconde_Depol,
	Minute_Restant=> Lect_Temp_Minute_Depol,
	Heure_Restant=> Lect_Temp_heure_Depol);

IF(RS_Depollution.Q1) // Version démarrage en manuel
	THEN
	Mode_Cabine_Depollution := TRUE;
	Sel_Etats_Cabine := 4;
	ELSE
	Mode_Cabine_Depollution := FALSE;
END_IF;

// Démarrage du premier cycle de dépollution qui nettoie la CTA pendant 5 minutes. Uniquement si utilisation de la CTA dans la recette
RS_CTA(SET:= (Mode_Cabine_Automatique AND RS_MEnCond.Q1), RESET1:= Mode_Cabine_Libre); // Détection du démarrage de la CTA
R_TRIG_cylcle1(CLK:= (Mode_Auto.Mode_10 AND RS_CTA.Q1)); // Démarrage via la recette, 1er cycle
TP_Cycle1(IN:= R_TRIG_cylcle1.Q, PT:= T#300S);
Mode_Depollution_cycle1 := TP_Cycle1.Q;

IF(Mode_Auto.Mode_10) // Démarrage via la recette 2ème cycle
	THEN
	Mode_Cabine_Depollution := TRUE;
END_IF;

(**************************************************************Gestion etat cabine nettoyage*)
IF(Start_Etat_Nettoyage AND NOT Mode_Cabine_Automatique AND NOT Mode_Cabine_Manuel AND NOT Mode_Cabine_Depollution  AND NOT Mode_Maintenance)
	THEN
	Mode_Cabine_Nettoyage := TRUE;
	Sel_Etats_Cabine := 5;
	ELSE
	Mode_Cabine_Nettoyage := FALSE;
END_IF;

(***************************************************************Gestion etat cabine Manuel*)
(*Mode arrêt du mode manuel*)
Mode_END_Manu := Mode_Arret_Manu;
(*Sécurité pour éviter de démarrer le mode manuel sans avoir réglé une consigne de temps supérieure à zéro*)
Securite_Tempo_Manu := Manu_Tempo_Transition_Seconde + Manu_Tempo_Transition_Minute + Manu_Tempo_Transition_Heure;

RS_Manu(SET:=
(Start_Mode_Manu AND NOT Mode_Cabine_Automatique AND (Securite_Tempo_Manu <> 0)),
RESET1:= Mode_END_Manu OR Mode_Cabine_Automatique OR Mode_Maintenance,
Q1=> Mode_Cabine_Manuel);

IF(Mode_Cabine_Manuel)
	THEN
	Sel_Etats_Cabine := 2;
END_IF;

(****************************************************************Gestion etat cabine Automatique*)
(*Mode arrêt du mode automatique*)
R_TRIG_FIN(CLK:= (Numero_Mode_Auto=0));
Mode_END_Auto := R_TRIG_FIN.Q;

RS_Automatique(
SET:= ((Start_Recette_Mode_Auto AND (Nbre_Etape_Totale <> 0))),
RESET1:= Mode_END_Auto OR Mode_Maintenance,
Q1=> Mode_Cabine_Automatique);

IF(Mode_Cabine_Automatique)
	THEN
	Sel_Etats_Cabine := 3;
END_IF;

(*****************************************************************Gestion etat cabine libre*)
IF((NOT Mode_Cabine_Manuel AND NOT Mode_Cabine_Automatique AND NOT Mode_Cabine_Depollution AND NOT Mode_Cabine_Nettoyage
			AND NOT Mode_Maintenance))
	THEN
	Sel_Etats_Cabine := 1;
	Mode_Cabine_Libre := TRUE;
	ELSE
	Mode_Cabine_Libre := FALSE;
END_IF;

(*****************************************************************Gestion etat cabine Maintenance*)
IF(Cmd_Mode_Maintenance)
	THEN
	Sel_Etats_Cabine := 7;
	Mode_Maintenance := TRUE;
	ELSE
	Mode_Maintenance := FALSE;
END_IF;

END_PROGRAM

// ---- POUs/Block/Autres/TON_V1.TcPOU
FUNCTION_BLOCK TON_V1
VAR_INPUT
	Enable: BOOL;
	Pause: BOOL;
	In_Cons_Seconde: REAL;
	In_Cons_Minute: REAL;
	In_Cons_Heure: REAL;
	In_Cons_Jour: REAL;
END_VAR
VAR_OUTPUT
	Q: BOOL;
	Seconde_Restant: REAL;
	Minute_Restant: REAL;
	Heure_Restant: REAL;
	Jour_Restant: REAL;
END_VAR
VAR
	TON_Inc: TON;
	R_TRIG_Inc: R_TRIG;
	Incrementation_Sec: BOOL;
	Valeur_Seconde: REAL;
	Valeur_Minutes: REAL;
	Valeur_Heures: REAL;
	Valeur_Jour: REAL;
	Var1: REAL;
	Var2: REAL;
	Var3: REAL;
	Var4: REAL;
	Seconde: REAL;
	Seconde_tot_Restant: REAL;
END_VAR

(*Comptage des secondes*)
TON_Inc(IN:= (NOT Incrementation_Sec AND NOT Pause AND NOT Q), PT:= T#1s, Q=> Incrementation_Sec );
R_TRIG_Inc(CLK:= Incrementation_Sec);

IF(Enable)
	THEN
(***************************************Comptage des secondes***************************************)
	IF(R_TRIG_Inc.Q AND NOT Q)
		THEN
		Valeur_Seconde := Valeur_Seconde + 1.0;
		Seconde := Seconde + 1.0;
	END_IF;
(****************************************Comptage des minutes****************************************)
	IF((Valeur_Seconde >= 60.0)  AND NOT Q)
		THEN
		Valeur_Seconde := 0.0;
		Valeur_Minutes := Valeur_Minutes + 1.0;
	END_IF;
(****************************************Comptage des heures****************************************)
	IF((Valeur_Minutes >= 60.0)   AND NOT Q)
		THEN
		Valeur_Minutes := 0.0;
		Valeur_Heures := Valeur_Heures + 1.0;
	END_IF;
(****************************************Comptage des jours****************************************)
	IF((Valeur_Heures >= 24.0) AND NOT Q)
		THEN
		Valeur_Heures := 0.0;
		Valeur_Jour := Valeur_Jour + 1.0;
	END_IF;
(****************************************Lors de l'arrêt****************************************)
	ELSE
	Var1 := 0.0;
	Var2 := 0.0;
	Var3 := 0.0;
	Var4 := 0.0;

	Valeur_Seconde := 0.0;
	Valeur_Minutes := 0.0;
	Valeur_Heures := 0.0;
	Valeur_Jour := 0.0;
	Seconde := 0.0;
	Seconde_tot_Restant := 0.0;
	Minute_Restant := 0;
	Heure_Restant := 0;
	Jour_Restant := 0;
	Q := FALSE;
END_IF;

(****************************************Calcul du temp restant****************************************)
Var1 := In_Cons_Minute * 60.0;
Var2 := In_Cons_Heure * 3600.0;
Var3 := In_Cons_Jour * 86400.0;
Var4 := Var1 + Var2 + Var3 + In_Cons_Seconde;

Seconde_tot_Restant := LIMIT(0, (Var4 - Seconde), 3000000);

Seconde_Restant := (REAL_TO_INT(Seconde_tot_Restant)) MOD 60;
Minute_Restant := (REAL_TO_INT(Seconde_tot_Restant) / 60) MOD 60;
Heure_Restant := (REAL_TO_INT(Seconde_tot_Restant) / 3600) MOD 24;
Jour_Restant := (REAL_TO_INT(Seconde_tot_Restant) / 86400) MOD 24;

(****************************************Sortie****************************************)
IF(Seconde >= (Var4 + 1) AND Enable)
	THEN
	Q := TRUE;
	ELSE
	Q := FALSE;
END_IF;

END_FUNCTION_BLOCK

// ---- POUs/g_Gestion_Texte_Modes.TcPOU
PROGRAM g_Gestion_Texte_Modes
VAR
	i: INT;
END_VAR

(*Gestion de l'affichage des noms de mode du protocole sélectionné*)
FOR i:=1 TO 29 BY 1 DO
	MEMSET(ADR(Tab_Nom_Mode[2,i]),0,SIZEOF(Tab_Nom_Mode[2,i]));
	IF (Tab_Recette_Auto[Numero_Recette_Sel, i,1] = 0) THEN Tab_Nom_Mode[2,i]:=''; END_IF;
	IF (Tab_Recette_Auto[Numero_Recette_Sel, i,1] = 1) THEN Tab_Nom_Mode[2,i]:='SHOWER WITH DRAIN AND DELAY'; END_IF;
	IF (Tab_Recette_Auto[Numero_Recette_Sel, i,1] = 2) THEN Tab_Nom_Mode[2,i]:='SHOWER WITHOUT DRAIN AND DELAY';  END_IF;
	IF (Tab_Recette_Auto[Numero_Recette_Sel, i,1] = 3) THEN Tab_Nom_Mode[2,i]:='CLEAN UP';  END_IF;
	IF (Tab_Recette_Auto[Numero_Recette_Sel, i,1] = 4) THEN Tab_Nom_Mode[2,i]:='SINK WITH DRAIN AND DELAY';  END_IF;
	IF (Tab_Recette_Auto[Numero_Recette_Sel, i,1] = 5) THEN Tab_Nom_Mode[2,i]:='SINK WITHOUT DRAIN AND DELAY';  END_IF;
	IF (Tab_Recette_Auto[Numero_Recette_Sel, i,1] = 6) THEN Tab_Nom_Mode[2,i]:='PLUG ACTIVATE';  END_IF;
	IF (Tab_Recette_Auto[Numero_Recette_Sel, i,1] = 7) THEN Tab_Nom_Mode[2,i]:='OPENED DRAIN';  END_IF;
	IF (Tab_Recette_Auto[Numero_Recette_Sel, i,1] = 8) THEN Tab_Nom_Mode[2,i]:='NEUTRAL';  END_IF;
	IF (Tab_Recette_Auto[Numero_Recette_Sel, i,1] = 9) THEN Tab_Nom_Mode[2,i]:='LARGE VOLUME TOILET FLUSH';  END_IF;
	IF (Tab_Recette_Auto[Numero_Recette_Sel, i,1] = 10) THEN Tab_Nom_Mode[2,i]:='DECONTAMINATION';  END_IF;
	IF (Tab_Recette_Auto[Numero_Recette_Sel, i,1] = 11) THEN Tab_Nom_Mode[2,i]:='NEUTRAL WITH LOW FLOW';  END_IF;
	IF (Tab_Recette_Auto[Numero_Recette_Sel, i,1] = 12) THEN Tab_Nom_Mode[2,i]:='SHOWER WITH DRAIN AND VOLUME'; END_IF;
	IF (Tab_Recette_Auto[Numero_Recette_Sel, i,1] = 13) THEN Tab_Nom_Mode[2,i]:='SHOWER WITHOUT DRAIN AND VOLUME';  END_IF;
	IF (Tab_Recette_Auto[Numero_Recette_Sel, i,1] = 14) THEN Tab_Nom_Mode[2,i]:='SINK WITH DRAIN AND VOLUME';  END_IF;
	IF (Tab_Recette_Auto[Numero_Recette_Sel, i,1] = 15) THEN Tab_Nom_Mode[2,i]:='SINK WITHOUT DRAIN AND VOLUME';  END_IF;
	IF (Tab_Recette_Auto[Numero_Recette_Sel, i,1] = 16) THEN Tab_Nom_Mode[2,i]:='SHOWER WITH DRAIN AND BUTTON'; END_IF;
	IF (Tab_Recette_Auto[Numero_Recette_Sel, i,1] = 17) THEN Tab_Nom_Mode[2,i]:='SINK WITH DRAIN AND BUTTON'; END_IF;
	IF (Tab_Recette_Auto[Numero_Recette_Sel, i,1] = 18) THEN Tab_Nom_Mode[2,i]:='HOT CLEANING'; END_IF;
	IF (Tab_Recette_Auto[Numero_Recette_Sel, i,1] = 19) THEN Tab_Nom_Mode[2,i]:='COLD CLEANING'; END_IF;
	IF (Tab_Recette_Auto[Numero_Recette_Sel, i,1] = 20) THEN Tab_Nom_Mode[2,i]:='PARAMETER MODE';  END_IF;
	IF (Tab_Recette_Auto[Numero_Recette_Sel, i,1] = 21) THEN Tab_Nom_Mode[2,i]:='PREPARATOR ALERT';  END_IF;
	IF (Tab_Recette_Auto[Numero_Recette_Sel, i,1] = 22) THEN Tab_Nom_Mode[2,i]:='EVALUATOR ALERT';  END_IF;
	IF (Tab_Recette_Auto[Numero_Recette_Sel, i,1] = 23) THEN Tab_Nom_Mode[2,i]:='EVALUATION';  END_IF;
	IF (Tab_Recette_Auto[Numero_Recette_Sel, i,1] = 24) THEN Tab_Nom_Mode[2,i]:='EVALUATION WITH AIR FLOW';  END_IF;
	IF (Tab_Recette_Auto[Numero_Recette_Sel, i,1] = 25) THEN Tab_Nom_Mode[2,i]:='CONDITIONING BOOTH';  END_IF;
	IF (Tab_Recette_Auto[Numero_Recette_Sel, i,1] = 26) THEN Tab_Nom_Mode[2,i]:='SMALL VOLUME TOILET FLUSH';  END_IF;
	IF (Tab_Recette_Auto[Numero_Recette_Sel, i,1] = 27) THEN Tab_Nom_Mode[2,i]:='CLEANING';  END_IF;
	IF (Tab_Recette_Auto[Numero_Recette_Sel, i,1] = 28) THEN Tab_Nom_Mode[2,i]:='BOOTH IN CONDITION';  END_IF;
	IF ((Tab_Recette_Auto[Numero_Recette_Sel, i,1] >= 30) AND (Tab_Recette_Auto[Numero_Recette_Sel, i,1] <= 59)) THEN Tab_Nom_Mode[2,i]:='USER MESSAGE';  END_IF;
	IF (Tab_Recette_Auto[Numero_Recette_Sel, i,1] = 99) THEN Tab_Nom_Mode[2,i]:='END MODE';  END_IF;

	MEMSET(ADR(Tab_Nom_Mode[1,i]),0,SIZEOF(Tab_Nom_Mode[1,i]));
	IF (Tab_Recette_Auto[Numero_Recette_Sel, i,1] = 0) THEN Tab_Nom_Mode[1,i]:='';  END_IF;
	IF (Tab_Recette_Auto[Numero_Recette_Sel, i,1] = 1) THEN Tab_Nom_Mode[1,i]:='DOUCHE BONDE OUVERTE ET TEMPO';  END_IF;
	IF (Tab_Recette_Auto[Numero_Recette_Sel, i,1] = 2) THEN Tab_Nom_Mode[1,i]:='DOUCHE BONDE FERMEE ET TEMPO';  END_IF;
	IF (Tab_Recette_Auto[Numero_Recette_Sel, i,1] = 3) THEN Tab_Nom_Mode[1,i]:='DOUCHETTE';  END_IF;
	IF (Tab_Recette_Auto[Numero_Recette_Sel, i,1] = 4) THEN Tab_Nom_Mode[1,i]:='LAVABO BONDE OUVERTE ET TEMPO';  END_IF;
	IF (Tab_Recette_Auto[Numero_Recette_Sel, i,1] = 5) THEN Tab_Nom_Mode[1,i]:='LAVABO BONDE FERMEE ET TEMPO';  END_IF;
	IF (Tab_Recette_Auto[Numero_Recette_Sel, i,1] = 6) THEN Tab_Nom_Mode[1,i]:='PRISE ELECTRIQUE';  END_IF;
	IF (Tab_Recette_Auto[Numero_Recette_Sel, i,1] = 7) THEN Tab_Nom_Mode[1,i]:='VIDANGE(S)';  END_IF;
	IF (Tab_Recette_Auto[Numero_Recette_Sel, i,1] = 8) THEN Tab_Nom_Mode[1,i]:='NEUTRE';  END_IF;
	IF (Tab_Recette_Auto[Numero_Recette_Sel, i,1] = 9) THEN Tab_Nom_Mode[1,i]:='CHASSE D EAU GRAND VOLUME';  END_IF;
	IF (Tab_Recette_Auto[Numero_Recette_Sel, i,1] = 10) THEN Tab_Nom_Mode[1,i]:='DEPOLLUTION';  END_IF;
	IF (Tab_Recette_Auto[Numero_Recette_Sel, i,1] = 11) THEN Tab_Nom_Mode[1,i]:='NEUTRE AVEC BAS DEBIT';  END_IF;
	IF (Tab_Recette_Auto[Numero_Recette_Sel, i,1] = 12) THEN Tab_Nom_Mode[1,i]:='DOUCHE BONDE OUVERTE ET VOLUME';  END_IF;
	IF (Tab_Recette_Auto[Numero_Recette_Sel, i,1] = 13) THEN Tab_Nom_Mode[1,i]:='DOUCHE BONDE FERMEE ET VOLUME';  END_IF;
	IF (Tab_Recette_Auto[Numero_Recette_Sel, i,1] = 14) THEN Tab_Nom_Mode[1,i]:='LAVABO BONDE OUVERTE ET VOLUME';  END_IF;
	IF (Tab_Recette_Auto[Numero_Recette_Sel, i,1] = 15) THEN Tab_Nom_Mode[1,i]:='LAVABO BONDE FERMEE ET VOLUME';  END_IF;
	IF (Tab_Recette_Auto[Numero_Recette_Sel, i,1] = 16) THEN Tab_Nom_Mode[1,i]:='DOUCHE BONDE OUVERTE ET BOUTON';  END_IF;
	IF (Tab_Recette_Auto[Numero_Recette_Sel, i,1] = 17) THEN Tab_Nom_Mode[1,i]:='LAVABO BONDE OUVERTE ET BOUTON';  END_IF;
	IF (Tab_Recette_Auto[Numero_Recette_Sel, i,1] = 18) THEN Tab_Nom_Mode[1,i]:='LAVAGE CHAUD';  END_IF;
	IF (Tab_Recette_Auto[Numero_Recette_Sel, i,1] = 19) THEN Tab_Nom_Mode[1,i]:='LAVAGE FROID';  END_IF;
	IF (Tab_Recette_Auto[Numero_Recette_Sel, i,1] = 20) THEN Tab_Nom_Mode[1,i]:='MODE PARAMETRABLE';  END_IF;
	IF (Tab_Recette_Auto[Numero_Recette_Sel, i,1] = 21) THEN Tab_Nom_Mode[1,i]:='ALERTE PREPARATEUR';  END_IF;
	IF (Tab_Recette_Auto[Numero_Recette_Sel, i,1] = 22) THEN Tab_Nom_Mode[1,i]:='ALERTE EVALUATEUR';  END_IF;
	IF (Tab_Recette_Auto[Numero_Recette_Sel, i,1] = 23) THEN Tab_Nom_Mode[1,i]:='EVALUATION';  END_IF;
	IF (Tab_Recette_Auto[Numero_Recette_Sel, i,1] = 24) THEN Tab_Nom_Mode[1,i]:='EVALUATION AVEC AIR';  END_IF;
	IF (Tab_Recette_Auto[Numero_Recette_Sel, i,1] = 25) THEN Tab_Nom_Mode[1,i]:='MISE EN CONDITION';  END_IF;
	IF (Tab_Recette_Auto[Numero_Recette_Sel, i,1] = 26) THEN Tab_Nom_Mode[1,i]:='CHASSE D EAU PETIT VOLUME';  END_IF;
	IF (Tab_Recette_Auto[Numero_Recette_Sel, i,1] = 27) THEN Tab_Nom_Mode[1,i]:='LAVAGE NEP';  END_IF;
	IF (Tab_Recette_Auto[Numero_Recette_Sel, i,1] = 28) THEN Tab_Nom_Mode[1,i]:='CABINE EN CONDITION';  END_IF;
	IF ((Tab_Recette_Auto[Numero_Recette_Sel, i,1] >= 30) AND (Tab_Recette_Auto[Numero_Recette_Sel, i,1] <= 59)) THEN Tab_Nom_Mode[1,i]:='MESSAGE UTILISATEUR';   END_IF;
	IF (Tab_Recette_Auto[Numero_Recette_Sel, i,1] = 99) THEN Tab_Nom_Mode[1,i]:='MODE FIN'; END_IF;
END_FOR;

(*Gestion d'écriture de la recette en cours de fonctionement*)
IF (Mode_Cabine_Automatique)
	THEN
	MEMSET(ADR(Tab_Nom_Recette[1,0]),0,SIZEOF(Tab_Nom_Recette[1,0]));
	MEMSET(ADR(Tab_Nom_Recette[2,0]),0,SIZEOF(Tab_Nom_Recette[2,0]));
	IF (Numero_Recette_Sel = 0)
		THEN
		Tab_Nom_Recette[1,0] := 'Recette en cours';
		Tab_Nom_Recette[2,0] := 'Protocol in progress';
		ELSE
		Tab_Nom_Recette[1,0] := Tab_Nom_Recette[1,Numero_Recette_Sel];
		Tab_Nom_Recette[2,0] := Tab_Nom_Recette[2,Numero_Recette_Sel];
	END_IF;
	ELSE
	MEMSET(ADR(Tab_Nom_Recette[1,0]),0,SIZEOF(Tab_Nom_Recette[1,0]));
	MEMSET(ADR(Tab_Nom_Recette[2,0]),0,SIZEOF(Tab_Nom_Recette[2,0]));
	Tab_Nom_Recette[1,0] := '';
	Tab_Nom_Recette[2,0] := '';
END_IF;

END_PROGRAM

// ---- POUs/Block/Cabines/Mode.TcPOU
FUNCTION_BLOCK Mode
VAR_INPUT
	Enable: BOOL;
	Numero_Etape: REAL;		(*Numéro de l'étape*)

(*Paramètre du tableau*)
	Numero_Mode: REAL;		(*Numéro du mode*)
	Tempo_Transition_seconde: REAL;
	Tempo_Transition_Minute: REAL;
	Tempo_Transition_Heure : REAL;
	Cons_Volume_Eau_Douche: REAL;
	Cons_Volume_Eau_Lavabo: REAL;
	Cons_Deb_Soufflage: REAL;
	Cons_Deb_Extraction: REAL;
	Cons_Temperature_Eau: REAL;
	Cons_Nbre_Chasse: REAL;
	Cons_Para_11: REAL;
	Cons_Para_12: REAL;
	Cons_Para_13: REAL;
	Cons_Para_14: REAL;
	Cons_Para_15: REAL;

END_VAR
VAR_OUTPUT
	Cmd_Douche: BOOL;
	Cmd_Lavabo: BOOL;
	Cmd_Douchette: BOOL;
	Cmd_NEP: BOOL;
	Cmd_Vidange_Douche: BOOL;
	Cmd_Vidange_Lavabo: BOOL;
	Cmd_Electrovanne_Douche :BOOL;
	Cmd_Electrovanne_Lavabo :BOOL;
	Cmd_Prise: BOOL;
	Cmd_Verin_WC_GV: BOOL;
	Cmd_Verin_WC_PV: BOOL;

	Out_Texte_FR: STRING(139);
	Out_Texte_ENG: STRING(139);

	Out_Cons_Moteur_ByPass: REAL;
	Out_Cons_V3V_Eau_Mitig: REAL;

	Out_Restant_Seconde: REAL;
	Out_Restant_Minute: REAL;
	Out_Restant_Heure: REAL;

	Out_Volume_Eau_Douche: REAL;
	Out_Volume_Eau_Lavabo: REAL;
	Out_Debit_Souf: REAL;
	Out_Debit_Ext: REAL;
	Out_Temp_Eau: REAL;
	Out_Para_11: REAL;
	Out_Para_12: REAL;
	Out_Para_13: REAL;
	Out_Para_14: REAL;
	Out_Para_15: REAL;

	Fin_Action: BOOL;
	Mode_END: BOOL;
END_VAR
VAR
(****************Autres****************)
	TON_Secu_Douche: TON;
	Temp_Secu_Douche: TIME;
	TON_Secu_Lavabo: TON;
	Temp_Secu_Lavabo: TIME;
	Secu_Volume_Douche: BOOL;
	Securite_Debord_Douche_Debit: BOOL;
	Secu_Volume_Lavabo: BOOL;
	Securite_Debord_Lavabo_Debit: BOOL;
	RS_Fin_Mode_1: RS;
	RS_Fin_Mode_2: RS;
	RS_Fin_Mode_4: RS;
	RS_Fin_Mode_5: RS;
	RS_Fin_Mode_7: RS;
	RS_Fin_Mode_18: RS;
	RS_Fin_Mode_19: RS;
	RS_Fin_Mode_27: RS;

	Cpt_Chasse_GV: REAL;
	Restart_Chasse_GV: BOOL;
	Tp_ChasseEau_GV: TP;
	Etp_Suiv_ChasseEau_GV: BOOL;
	R_TRIG_Cpt_Chasse_GV: R_TRIG;

	Cpt_Chasse_PV: REAL;
	Restart_Chasse_PV: BOOL;
	Tp_ChasseEau_PV: TP;
	Etp_Suiv_ChasseEau_PV: BOOL;
	R_TRIG_Cpt_Chasse_PV: R_TRIG;
(****************Mode avec temporisation****************)
	TON_Mode1: TON_V1;
	Mode_1: BOOL;
	TON_Mode2: TON_V1;
	Mode_2: BOOL;
	TON_Mode4: TON_V1;
	Mode_4: BOOL;
	TON_Mode5: TON_V1;
	Mode_5: BOOL;
	TON_Mode6: TON_V1;
	Mode_6: BOOL;
	TON_Mode7: TON_V1;
	Mode_7: BOOL;
	TON_Mode8: TON_V1;
	Mode_8: BOOL;
	TON_Mode9: TON_V1;
	Mode_9: BOOL;
	TON_Mode10: TON_V1;
	Mode_10: BOOL;
	TON_Mode11: TON_V1;
	Mode_11: BOOL;
	TON_Mode18: TON_V1;
	Mode_18: BOOL;
	TON_Mode19: TON_V1;
	Mode_19: BOOL;
	TON_Mode21: TON;
	Mode_21: BOOL;
	TON_Mode22: TON;
	Mode_22: BOOL;
	TON_Mode26: TON_V1;
	Mode_26: BOOL;
	TON_Mode27: TON_V1;
	Mode_27: BOOL;
(****************Mode Texte avec validation****************)
	Mode_3: BOOL;
	F_TRIG_Texte3: F_TRIG;
	Mode_23: BOOL;
	F_TRIG_Texte23: F_TRIG;
	Mode_30: BOOL;
	F_TRIG_Texte30: F_TRIG;
	Mode_16: BOOL;
	F_TRIG_Texte16: F_TRIG;
	Mode_17: BOOL;
	F_TRIG_Texte17: F_TRIG;
	Mode_24: BOOL;
	F_TRIG_Texte24: F_TRIG;
(****************Mode Gestion volume****************)
	Mode_12 :BOOL;
	Integr_Vol_Eau_Mode12: Integr_Vol_Eau;
	R_TRIG_Mode12: R_TRIG;
	Calcul_Offset_Mode12: REAL;
	Mode_13 :BOOL;
	Integr_Vol_Eau_Mode13: Integr_Vol_Eau;
	R_TRIG_Mode13: R_TRIG;
	Calcul_Offset_Mode13: REAL;
	Mode_14 :BOOL;
	Integr_Vol_Eau_Mode14: Integr_Vol_Eau;
	R_TRIG_Mode14: R_TRIG;
	Calcul_Offset_Mode14: REAL;
	Mode_15 :BOOL;
	Integr_Vol_Eau_Mode15: Integr_Vol_Eau;
	R_TRIG_Mode15: R_TRIG;
	Calcul_Offset_Mode15: REAL;
(****************Pour enceinte climatique****************)
	Mode_25: BOOL;
	F_TRIG_Mode25: F_TRIG;
	TON_Temp_Ok: TON;
	Temp_Ok: BOOL;
	TON_Hygro_Ok: TON;
	Hygro_Ok: BOOL;
	Validation_Temp_Hygro: BOOL;
	TP_RAZ_Mode25: TP;
	R_TRIG_Valide_TempHygro: R_TRIG;
	Mode_28: BOOL;
	F_TRIG_Mode28: F_TRIG;
END_VAR

MEMSET(ADR(Out_Texte_FR),0,SIZEOF(Out_Texte_FR));
MEMSET(ADR(Out_Texte_ENG),0,SIZEOF(Out_Texte_ENG));

(****************************************************************Mode 1 : Mode douche avec vidange transition temporisation****************************************************************)
Mode_1 := Numero_Mode = 1 AND Enable;
IF(Mode_1  AND NOT Fin_Action)
	THEN
	(*Gestion du texte*)
	IF(E_Vanne_Vidange_Douche_Ouv)
		THEN
		Out_Texte_FR := 'DOUCHE BONDE OUVERTE ET TEMPO';
		Out_Texte_ENG := 'SHOWER WITH DRAIN AND DELAY';
		ELSE
		Out_Texte_FR := 'DOUCHE BONDE OUVERTE ET TEMPO - OUVERTURE BONDE';
		Out_Texte_ENG :=  'SHOWER WITH DRAIN AND DELAY - OPENING DRAIN';
	END_IF;
	IF(RS_Fin_Mode_1.Q1)
		THEN
		Out_Texte_FR := 'DOUCHE BONDE OUVERTE ET TEMPO - FERMETURE DOUCHE';
		Out_Texte_ENG := 'SHOWER WITH DRAIN AND DELAY - CLOSING SHOWER';
	END_IF;

	(*Gestion de la commande de la douche et de la vidange*)
	Cmd_Vidange_Douche := TRUE;
	IF( RS_Fin_Mode_1.Q1)
		THEN
		Out_Restant_Seconde := 0.0;
		Out_Restant_Minute := 0.0;
		Out_Restant_Heure := 0.0;
		Cmd_Douche := FALSE;
		ELSE
		IF(E_Vanne_Vidange_Douche_Ouv)
			THEN
			Cmd_Douche := TRUE;
			Cmd_Electrovanne_Douche := TRUE;
			ELSE
			Cmd_Douche := FALSE;
			Cmd_Electrovanne_Douche := FALSE;
		END_IF;
	END_IF;

	(*Gestion de la commande pause*)
	IF(Comande_Pause)
		THEN
		Cmd_Douche := FALSE;
		Cmd_Electrovanne_Douche := FALSE;
	END_IF;

	(*Gestion du décompte de la temporisation du mode*)
	Out_Restant_Seconde := TON_Mode1.Seconde_Restant;
	Out_Restant_Minute := TON_Mode1.Minute_Restant;
	Out_Restant_Heure := TON_Mode1.Heure_Restant;

	(*Gestion des lectures consignes du mode*)
	Out_Debit_Souf 			:= Cons_Deb_Soufflage;
	Out_Debit_Ext 			:= Cons_Deb_Extraction;
	Out_Temp_Eau 			:= Cons_Temperature_Eau;

	(*Initialisation des actionneurs non utilisés*)
	Cmd_Lavabo := FALSE;
	Cmd_Douchette := FALSE;
	Cmd_NEP := FALSE;
	Cmd_Vidange_Lavabo := FALSE;
	Cmd_Electrovanne_Lavabo := FALSE;
	Cmd_Prise := FALSE;
	Cmd_Verin_WC_GV := FALSE;
	Cmd_Verin_WC_PV := FALSE;
END_IF;
(*************************************Temporisation du décompte du mode*************************************)
TON_Mode1(
Enable:= (Mode_1 AND (E_Vanne_Vidange_Douche_Ouv OR Comande_Pause)),
Pause:= Comande_Pause,
In_Cons_Seconde:= Tempo_Transition_Seconde,
In_Cons_Minute:= Tempo_Transition_Minute,
In_Cons_Heure:= Tempo_Transition_Heure);

(*Activation de la fin du mode*)
RS_Fin_Mode_1(SET:= TON_Mode1.Q, RESET1:= NOT Mode_1);
IF( RS_Fin_Mode_1.Q1)
	THEN
	Out_Restant_Seconde := 0.0;
	Out_Restant_Minute := 0.0;
	Out_Restant_Heure := 0.0;
END_IF;

(***************************************************************Mode 2 : Mode douche sans vidange transition temporisation****************************************************************)
Mode_2 := Numero_Mode = 2 AND Enable;
IF(Mode_2  AND NOT Fin_Action)
	THEN
	(*Gestion du texte*)
	IF(E_Vanne_Vidange_Douche_Ferm)
		THEN
		Out_Texte_FR := 'DOUCHE BONDE FERMEE ET TEMPO';
		Out_Texte_ENG := 'SHOWER WITHOUT DRAIN AND DELAY';
		ELSE
		Out_Texte_FR := 'DOUCHE BONDE FERMEE ET TEMPO - FERMETURE BONDE';
		Out_Texte_ENG := 'SHOWER WITHOUT DRAIN AND DELAY - CLOSING DRAIN';
	END_IF;
	IF(RS_Fin_Mode_2.Q1)
		THEN
		Out_Texte_FR := 'DOUCHE BONDE FERMEE ET TEMPO - FERMETURE DOUCHE';
		Out_Texte_ENG := 'SHOWER WITHOUT DRAIN AND DELAY - CLOSING SHOWER';
	END_IF;

	(*Gestion de la commande de la douche*)
	Cmd_Vidange_Douche := FALSE;
	IF( RS_Fin_Mode_2.Q1)
		THEN
		Out_Restant_Seconde := 0.0;
		Out_Restant_Minute := 0.0;
		Out_Restant_Heure := 0.0;
		Cmd_Douche := FALSE;
		ELSE
		IF(E_Vanne_Vidange_Douche_Ferm)
			THEN
			Cmd_Douche := TRUE;
			Cmd_Electrovanne_Douche := TRUE;
			ELSE
			Cmd_Douche := FALSE;
			Cmd_Electrovanne_Douche := FALSE;
		END_IF;
	
		IF(Comande_Pause)
			THEN
			Cmd_Douche := FALSE;
			Cmd_Electrovanne_Douche := FALSE;
		END_IF;
	END_IF;

	(*Gestion du décompte de la temporisation du mode*)
	Out_Restant_Seconde := TON_Mode2.Seconde_Restant;
	Out_Restant_Minute := TON_Mode2.Minute_Restant;
	Out_Restant_Heure := TON_Mode2.Heure_Restant;

	(*Gestion des lectures consignes du mode*)
	Out_Debit_Souf 			:= Cons_Deb_Soufflage;
	Out_Debit_Ext 			:= Cons_Deb_Extraction;
	Out_Temp_Eau 			:= Cons_Temperature_Eau;

	(*Initialisation des actionneurs non utilisés*)
	Cmd_Lavabo := FALSE;
	Cmd_Douchette := FALSE;
	Cmd_NEP := FALSE;
	Cmd_Vidange_Douche := FALSE;
	Cmd_Vidange_Lavabo := FALSE;
	Cmd_Electrovanne_Lavabo := FALSE;
	Cmd_Prise := FALSE;
	Cmd_Verin_WC_GV := FALSE;
	Cmd_Verin_WC_PV := FALSE;
END_IF;

(*************************************Temporisation du décompte du mode*************************************)
TON_Mode2(
	Enable:= (Mode_2 AND ((E_Vanne_Vidange_Douche_Ferm) OR Comande_Pause)),
	Pause:= Comande_Pause,
	In_Cons_Seconde:= Tempo_Transition_Seconde,
	In_Cons_Minute:= Tempo_Transition_Minute,
	In_Cons_Heure:= Tempo_Transition_Heure);

(*Activation de la fin du mode*)
RS_Fin_Mode_2(SET:= TON_Mode2.Q, RESET1:= NOT Mode_2);
IF( RS_Fin_Mode_2.Q1)
	THEN
	Out_Restant_Seconde := 0.0;
	Out_Restant_Minute := 0.0;
	Out_Restant_Heure := 0.0;
END_IF;

(****************************************************************Mode 3 : Mode douchette avec vidanges****************************************************************)
Mode_3 := Numero_Mode = 3 AND Enable;
(*Validation de l'étape suivante*)
F_TRIG_Texte3(CLK:= (Valid_Texte AND Mode_3));
IF(Mode_3 AND NOT Fin_Action)
	THEN
	(*Gestion du texte*)
	IF(E_Vanne_Vidange_Douche_Ouv OR E_Vanne_Alim_Lavabo_Ouv)
		THEN
		Out_Texte_FR := 'DOUCHETTE';
		Out_Texte_ENG := 'HANDSPRAY WITH DRAIN';
		ELSE
		Out_Texte_FR := 'DOUCHETTE - OUVERTURE BONDE';
		Out_Texte_ENG := 'HANDSPRAY WITH DRAIN - OPENING DRAIN';
	END_IF;

	(*Gestion de la commande de la douchette avec vidange douche et lavabo*)
	Cmd_Vidange_Douche := TRUE;
	Cmd_Vidange_Lavabo := TRUE;
	IF(E_Vanne_Vidange_Douche_Ouv OR E_Vanne_Alim_Lavabo_Ouv)
		THEN
		Cmd_Douchette := TRUE;
		ELSE
		Cmd_Douchette := FALSE;
	END_IF;

	IF(Comande_Pause)
		THEN
		Cmd_Douchette := FALSE;
	END_IF;

	(*Gestion des lectures consignes du mode*)
	Out_Debit_Souf 			:= Cons_Deb_Souf_Etat_Nettoyage;
	Out_Debit_Ext 			:= Cons_Deb_Souf_Etat_Nettoyage;
	Out_Temp_Eau 			:= Cons_Temperature_Eau;

	(*Initialisation des actionneurs non utilisés*)
	Cmd_Douche := FALSE;
	Cmd_Lavabo := FALSE;
	Cmd_NEP := FALSE;
	Cmd_Electrovanne_Douche := FALSE;
	Cmd_Electrovanne_Lavabo := FALSE;
	Cmd_Prise := FALSE;
	Cmd_Verin_WC_GV := FALSE;
	Cmd_Verin_WC_PV := FALSE;
END_IF;

(****************************************************************Mode 4 : Mode Lavabo avec vidange transition temporisation****************************************************************)
Mode_4 := Numero_Mode = 4 AND Enable;
IF(Mode_4 AND NOT Fin_Action)
	THEN
	(*Gestion du texte*)
	IF(E_Vanne_Vidange_Lavabo_Ouv)
		THEN
		Out_Texte_FR := 'LAVABO BONDE OUVERTE ET TEMPO';
		Out_Texte_ENG := 'SINK WITH DRAIN AND DELAY';
		ELSE
		Out_Texte_FR := 'LAVABO BONDE OUVERTE ET TEMPO - OUVERTURE BONDE';
		Out_Texte_ENG := 'SINK WITH DRAIN AND DELAY - OPENING DRAIN';
	END_IF;
	IF(RS_Fin_Mode_4.Q1)
		THEN
		Out_Texte_FR := 'LAVABO BONDE OUVERTE ET TEMPO - FERMETURE LAVABO';
		Out_Texte_ENG := 'SINK WITH DRAIN AND DELAY - CLOSING SINK';
	END_IF;

	(*Gestion de la commande du lavabo avec la vidange*)
	Cmd_Vidange_Lavabo := TRUE;
	IF( RS_Fin_Mode_4.Q1)
		THEN
		Out_Restant_Seconde := 0.0;
		Out_Restant_Minute := 0.0;
		Out_Restant_Heure := 0.0;
		Cmd_Lavabo := FALSE;
		ELSE
		IF(E_Vanne_Vidange_Lavabo_Ouv)
			THEN
			Cmd_Lavabo := TRUE;
			Cmd_Electrovanne_Lavabo := TRUE;
			ELSE
			Cmd_Lavabo := FALSE;
			Cmd_Electrovanne_Lavabo := FALSE;
		END_IF;
	
		IF(Comande_Pause)
			THEN
			Cmd_Lavabo := FALSE;
			Cmd_Electrovanne_Lavabo := FALSE;
		END_IF;
	END_IF;

	(*Gestion du décompte de la temporisation du mode*)
	Out_Restant_Seconde := TON_Mode4.Seconde_Restant;
	Out_Restant_Minute := TON_Mode4.Minute_Restant;
	Out_Restant_Heure := TON_Mode4.Heure_Restant;

	(*Gestion des lectures consignes du mode*)
	Out_Debit_Souf 			:= Cons_Deb_Soufflage;
	Out_Debit_Ext 			:= Cons_Deb_Extraction;
	Out_Temp_Eau 			:= Cons_Temperature_Eau;

	(*Initialisation des actionneurs non utilisés*)
	Cmd_Douche := FALSE;
	Cmd_Douchette := FALSE;
	Cmd_NEP := FALSE;
	Cmd_Vidange_Douche := FALSE;
	Cmd_Electrovanne_Douche := FALSE;
	Cmd_Prise := FALSE;
	Cmd_Verin_WC_GV := FALSE;
	Cmd_Verin_WC_PV := FALSE;
END_IF;
(*************************************Temporisation du décompte du mode*************************************)
TON_Mode4(
	Enable:= (Mode_4 AND (E_Vanne_Vidange_Lavabo_Ouv OR Comande_Pause)),
	Pause:= Comande_Pause,
	In_Cons_Seconde:= Tempo_Transition_Seconde,
	In_Cons_Minute:= Tempo_Transition_Minute,
	In_Cons_Heure:= Tempo_Transition_Heure);

(*Activation de la fin du mode*)
RS_Fin_Mode_4(SET:= TON_Mode4.Q, RESET1:= NOT Mode_4);
IF( RS_Fin_Mode_4.Q1)
	THEN
	Out_Restant_Seconde := 0.0;
	Out_Restant_Minute := 0.0;
	Out_Restant_Heure := 0.0;
END_IF;

(****************************************************************Mode 5 : Mode Lavabo sans vidange transition temporisation****************************************************************)
Mode_5 := Numero_Mode = 5 AND Enable;
IF(Mode_5 AND NOT Fin_Action)
	THEN
	(*Gestion du texte*)
	IF(E_Vanne_Vidange_Lavabo_Ferm)
		THEN
		Out_Texte_FR := 'LAVABO BONDE FERMEE ET TEMPO';
		Out_Texte_ENG := 'SINK WITHOUT DRAIN AND DELAY';
		ELSE
		Out_Texte_FR := 'LAVABO BONDE FERMEE ET TEMPO - FERMETURE BONDE';
		Out_Texte_ENG := 'SINK WITHOUT DRAIN AND DELAY - CLOSING DRAIN';
	END_IF;
	IF(RS_Fin_Mode_5.Q1)
		THEN
		Out_Texte_FR := 'LAVABO BONDE FERMEE ET TEMPO - FERMETURE LAVABO';
		Out_Texte_ENG := 'SINK WITHOUT DRAIN AND DELAY - CLOSING SINK';
	END_IF;

	(*Gestion de la commande du lavabo*)
	Cmd_Vidange_Lavabo := FALSE;
	IF( RS_Fin_Mode_5.Q1)
		THEN
		Out_Restant_Seconde := 0.0;
		Out_Restant_Minute := 0.0;
		Out_Restant_Heure := 0.0;
		Cmd_Lavabo := FALSE;
		ELSE
		IF(E_Vanne_Vidange_Lavabo_Ferm)
			THEN
			Cmd_Lavabo := TRUE;
			Cmd_Electrovanne_Lavabo := TRUE;
			ELSE
			Cmd_Lavabo := FALSE;
			Cmd_Electrovanne_Lavabo := FALSE;
		END_IF;
	
		IF(Comande_Pause)
			THEN
			Cmd_Lavabo := FALSE;
			Cmd_Electrovanne_Lavabo := FALSE;
		END_IF;
	END_IF;

	(*Gestion du décompte de la temporisation du mode*)
	Out_Restant_Seconde := TON_Mode5.Seconde_Restant;
	Out_Restant_Minute := TON_Mode5.Minute_Restant;
	Out_Restant_Heure := TON_Mode5.Heure_Restant;

	(*Gestion des lectures consignes du mode*)
	Out_Debit_Souf 			:= Cons_Deb_Soufflage;
	Out_Debit_Ext 			:= Cons_Deb_Extraction;
	Out_Temp_Eau 			:= Cons_Temperature_Eau;

	(*Initialisation des actionneurs non utilisés*)
	Cmd_Douche := FALSE;
	Cmd_Douchette := FALSE;
	Cmd_NEP := FALSE;
	Cmd_Vidange_Douche := FALSE;
	Cmd_Vidange_Lavabo := FALSE;
	Cmd_Electrovanne_Douche := FALSE;
	Cmd_Prise := FALSE;
	Cmd_Verin_WC_GV := FALSE;
	Cmd_Verin_WC_PV := FALSE;
END_IF;
(*************************************Temporisation du décompte du mode*************************************)
TON_Mode5(
	Enable:= (Mode_5 AND ((E_Vanne_Vidange_Lavabo_Ferm) OR Comande_Pause)),
	Pause:= Comande_Pause,
	In_Cons_Seconde:= Tempo_Transition_Seconde,
	In_Cons_Minute:= Tempo_Transition_Minute,
	In_Cons_Heure:= Tempo_Transition_Heure);

(*Activation de la fin du mode*)
RS_Fin_Mode_5(SET:= TON_Mode5.Q, RESET1:= NOT Mode_5);
IF( RS_Fin_Mode_5.Q1)
	THEN
	Out_Restant_Seconde := 0.0;
	Out_Restant_Minute := 0.0;
	Out_Restant_Heure := 0.0;
END_IF;

(****************************************************************Mode 6 : Mode activation prise****************************************************************)
Mode_6 := Numero_Mode = 6 AND Enable;
IF(Mode_6 AND NOT Fin_Action)
	THEN
	(*Gestion du texte*)
	Out_Texte_FR := 'PRISE ELECTRIQUE';
	Out_Texte_ENG := 'PLUG ACTIVATED';

	(*Gestion de la commande de la prise*)
	Cmd_Prise := TRUE;

	IF(Comande_Pause)
		THEN
		Cmd_Prise := TRUE;
	END_IF;

	(*Gestion du décompte de la temporisation du mode*)
	Out_Restant_Seconde := TON_Mode6.Seconde_Restant;
	Out_Restant_Minute := TON_Mode6.Minute_Restant;
	Out_Restant_Heure := TON_Mode6.Heure_Restant;

	(*Gestion des lectures consignes du mode*)
	Out_Debit_Souf 			:= Cons_Deb_Soufflage;
	Out_Debit_Ext 			:= Cons_Deb_Extraction;
	Out_Temp_Eau 			:= Cons_Temperature_Eau;

	(*Initialisation des actionneurs non utilisés*)
	Cmd_Douchette := FALSE;
	Cmd_Douche := FALSE;
	Cmd_Lavabo := FALSE;
	Cmd_NEP := FALSE;
	Cmd_Vidange_Douche := FALSE;
	//Cmd_Vidange_Lavabo := FALSE;
	Cmd_Verin_WC_GV := FALSE;
	Cmd_Verin_WC_PV := FALSE;
END_IF;
(*************************************Temporisation du décompte du mode*************************************)
TON_Mode6(
	Enable:= ((Mode_6 OR Comande_Pause)),
	Pause:= Comande_Pause,
	In_Cons_Seconde:= Tempo_Transition_Seconde,
	In_Cons_Minute:= Tempo_Transition_Minute,
	In_Cons_Heure:= Tempo_Transition_Heure);

(****************************************************************Mode 7 : Mode  vidanges****************************************************************)
Mode_7 := Numero_Mode = 7 AND Enable;
IF(Mode_7 AND NOT Fin_Action)
	THEN
	(*Gestion du texte*)
	IF(E_Vanne_Vidange_Douche_Ouv OR E_Vanne_Vidange_Lavabo_Ouv)
		THEN
		Out_Texte_FR := 'VIDANGE(S)';
		Out_Texte_ENG := 'DRAIN';
		ELSE
		Out_Texte_FR := 'VIDANGE(S) - OUVERTURE BONDE(S)';
		Out_Texte_ENG := 'DRAIN - OPENING DRAIN';
	END_IF;

	(*Gestion de la commande des vidanges douche et lavabo*)
	Cmd_Vidange_Douche := TRUE;
	Cmd_Vidange_Lavabo := TRUE;

	(*Gestion du décompte de la temporisation du mode*)
	Out_Restant_Seconde := TON_Mode7.Seconde_Restant;
	Out_Restant_Minute := TON_Mode7.Minute_Restant;
	Out_Restant_Heure := TON_Mode7.Heure_Restant;

	(*Gestion des lectures consignes du mode*)
	Out_Debit_Souf 			:= Cons_Deb_Soufflage;
	Out_Debit_Ext 			:= Cons_Deb_Extraction;
	Out_Temp_Eau 			:= Cons_Temperature_Eau;

	(*Initialisation des actionneurs non utilisés*)
	Cmd_Douche := FALSE;
	Cmd_Lavabo := FALSE;
	Cmd_Douchette := FALSE;
	Cmd_NEP := FALSE;
	Cmd_Electrovanne_Douche := FALSE;
	Cmd_Electrovanne_Lavabo := FALSE;
	Cmd_Prise := FALSE;
	Cmd_Verin_WC_GV := FALSE;
	Cmd_Verin_WC_PV := FALSE;
END_IF;
(*************************************Temporisation du décompte du mode*************************************)
TON_Mode7(
	Enable:= ((Mode_7 AND (E_Vanne_Vidange_Douche_Ouv AND E_Vanne_Vidange_Lavabo_Ouv AND Option_Douche AND Option_Lavabo) (*Option douche + Lavabo*)
			OR (E_Vanne_Vidange_Douche_Ouv AND Option_Douche AND NOT Option_Lavabo) (*Option douche*)
			OR (E_Vanne_Vidange_Lavabo_Ouv AND Option_Lavabo AND NOT Option_Douche)) (*Option lavabo*)
			OR Comande_Pause),
	Pause:= Comande_Pause,
	In_Cons_Seconde:= Tempo_Transition_Seconde,
	In_Cons_Minute:= Tempo_Transition_Minute,
	In_Cons_Heure:= Tempo_Transition_Heure);
(*Activation de la fin du mode*)
RS_Fin_Mode_7(SET:= TON_Mode7.Q, RESET1:= NOT Mode_7);
IF( RS_Fin_Mode_7.Q1)
	THEN
	Out_Restant_Seconde := 0.0;
	Out_Restant_Minute := 0.0;
	Out_Restant_Heure := 0.0;
END_IF;

(****************************************************************Mode 8 : Mode Neutre****************************************************************)
Mode_8 := Numero_Mode = 8 AND Enable;
IF(Mode_8 AND NOT Fin_Action)
	THEN
	(*Gestion du texte*)
	Out_Texte_FR := 'NEUTRE';
	Out_Texte_ENG := 'NEUTRAL';

	(*Gestion du décompte de la temporisation du mode*)
	Out_Restant_Seconde := TON_Mode8.Seconde_Restant;
	Out_Restant_Minute := TON_Mode8.Minute_Restant;
	Out_Restant_Heure := TON_Mode8.Heure_Restant;

	(*Gestion des lectures consignes du mode*)
	Out_Debit_Souf 			:= 0.0;
	Out_Debit_Ext 			:= 0.0;
	Out_Temp_Eau 			:= Cons_Temperature_Eau;

	(*Initialisation des actionneurs non utilisés*)
	Cmd_Douche := FALSE;
	Cmd_Lavabo := FALSE;
	Cmd_Douchette := FALSE;
	Cmd_NEP := FALSE;
	Cmd_Vidange_Douche := FALSE;
	//Cmd_Vidange_Lavabo := FALSE;
	Cmd_Electrovanne_Douche := FALSE;
	Cmd_Electrovanne_Lavabo := FALSE;
	Cmd_Prise := FALSE;
	Cmd_Verin_WC_GV := FALSE;
	Cmd_Verin_WC_PV := FALSE;
END_IF;
(*************************************Temporisation du décompte du mode*************************************)
TON_Mode8(
	Enable:= (Mode_8 OR Comande_Pause),
	Pause:= Comande_Pause,
	In_Cons_Seconde:= Tempo_Transition_Seconde,
	In_Cons_Minute:= Tempo_Transition_Minute,
	In_Cons_Heure:= Tempo_Transition_Heure);

(****************************************************************Mode 9 : Mode chasse d'eau Grand volume****************************************************************)
Mode_9 := Numero_Mode = 9 AND Enable;
IF(Mode_9 AND NOT Fin_Action)
	THEN
	(*Gestion du texte*)
	Out_Texte_FR := 'CHASSE D EAU GRAND VOLUME';
	Out_Texte_ENG := 'LARGE VOLUME TOILET FLUSH';

	(*Gestion du décompte de la temporisation du mode*)
	Out_Restant_Seconde := TON_Mode9.Seconde_Restant;
	Out_Restant_Minute := TON_Mode9.Minute_Restant;
	Out_Restant_Heure := TON_Mode9.Heure_Restant;

	(*Démarrage du premier cycle de chasse avant la temporisation*)
	R_TRIG_Cpt_Chasse_GV(CLK:= (Mode_9));

	(*Comptage du nombre de cycle x*)
	IF (TON_Mode9.Q OR R_TRIG_Cpt_Chasse_GV.Q)
		THEN
		Cpt_Chasse_GV := Cpt_Chasse_GV + 1;
		Restart_Chasse_GV := TRUE;
	END_IF;

	(*Initialisation des actionneurs non utilisés*)
	Cmd_Douche := FALSE;
	Cmd_Lavabo := FALSE;
	Cmd_Douchette := FALSE;
	Cmd_NEP := FALSE;
	Cmd_Electrovanne_Douche := FALSE;
	Cmd_Electrovanne_Lavabo := FALSE;
	Cmd_Prise := FALSE;
	Cmd_Verin_WC_PV := FALSE;
END_IF;
(*************************************Temporisation du décompte du mode*************************************)
TON_Mode9(
	Enable:= ((Mode_9 OR Comande_Pause OR Tp_ChasseEau_GV.Q) AND NOT Restart_Chasse_GV),
	Pause:= Comande_Pause OR Tp_ChasseEau_GV.Q,
	In_Cons_Seconde:= Tempo_Transition_Seconde,
	In_Cons_Minute:= Tempo_Transition_Minute,
	In_Cons_Heure:= Tempo_Transition_Heure);
Restart_Chasse_GV := FALSE;
(*Commande de la chasse d'eau pendant x secondes*)
Tp_ChasseEau_GV(IN:= TON_Mode9.Q OR R_TRIG_Cpt_Chasse_GV.Q, PT:= T#2s);
IF (Tp_ChasseEau_GV.Q AND Mode_9) THEN Cmd_Verin_WC_GV := TRUE; ELSE Cmd_Verin_WC_GV := FALSE; END_IF;
(*FIn du mode quand le nombre de cycle est atteint*)
IF ((Cpt_Chasse_GV >= Cons_Nbre_Chasse) AND Mode_9 AND NOT Tp_ChasseEau_GV.Q)
	THEN Etp_Suiv_ChasseEau_GV := TRUE; Cpt_Chasse_GV := 0.0;
	ELSE Etp_Suiv_ChasseEau_GV := FALSE; END_IF;

(****************************************************************Mode 10 : Mode Depollution****************************************************************)
Mode_10 := Numero_Mode = 10 AND Enable;
IF(Mode_10 AND NOT Fin_Action)
	THEN
	(*Gestion du texte*)
	Out_Texte_FR := 'DEPOLLUTION';
	Out_Texte_ENG := 'DECONTAMINATION';

	(*Gestion du décompte de la temporisation du mode*)
	Out_Restant_Seconde := TON_Mode10.Seconde_Restant;
	Out_Restant_Minute := TON_Mode10.Minute_Restant;
	Out_Restant_Heure := TON_Mode10.Heure_Restant;

	(*Gestion des lectures consignes du mode*)
	IF(Dmd_Post_Ventilation)
		THEN
		Out_Debit_Souf 			:= 0.0;
		Out_Debit_Ext 			:= 0.0;
		ELSE
		Out_Debit_Souf 			:= Cons_Deb_Souf_Etat_Depol;
		Out_Debit_Ext 			:= Cons_Deb_Souf_Etat_Depol;
	END_IF;
		Out_Volume_Eau_Douche 	:= Cons_Volume_Eau_Douche;
		Out_Volume_Eau_Lavabo 	:= Cons_Volume_Eau_Lavabo;
		Out_Temp_Eau 			:= Cons_Temperature_Eau;

	(*Initialisation des actionneurs non utilisés*)
	Cmd_Douche := FALSE;
	Cmd_Lavabo := FALSE;
	Cmd_Douchette := FALSE;
	Cmd_NEP := FALSE;
	Cmd_Electrovanne_Douche := FALSE;
	Cmd_Electrovanne_Lavabo := FALSE;
	Cmd_Prise := FALSE;
	Cmd_Verin_WC_GV := FALSE;
	Cmd_Verin_WC_PV := FALSE;
END_IF;
(*************************************Temporisation du décompte du mode*************************************)
TON_Mode10(
	Enable:= (Mode_10 OR Comande_Pause),
	Pause:= Comande_Pause,
	In_Cons_Seconde:= Tempo_Transition_Seconde,
	In_Cons_Minute:= Tempo_Transition_Minute,
	In_Cons_Heure:= Tempo_Transition_Heure);

(****************************************************************Mode 11 : Neutre avec bas débit****************************************************************)
Mode_11 := Numero_Mode = 11 AND Enable;
IF(Mode_11  AND NOT Fin_Action)
	THEN
	(*Gestion du texte*)
	IF(E_Vanne_Souf_Bas_Deb_Ouv AND E_Vanne_Ext_Bas_Deb_Ouv)
		THEN
		Out_Texte_FR := 'NEUTRE AVEC  BAS DEBIT';
		Out_Texte_ENG := 'NEUTRAL WITH LOW FLOW';
		ELSE
		Out_Texte_FR := 'NEUTRE AVEC  BAS DEBIT - OUVERTURE';
		Out_Texte_ENG :=  'SHOWER WITH DRAIN AND DELAY - OPENING';
	END_IF;

	(*Gestion du décompte de la temporisation du mode*)
	Out_Restant_Seconde := TON_Mode11.Seconde_Restant;
	Out_Restant_Minute := TON_Mode11.Minute_Restant;
	Out_Restant_Heure := TON_Mode11.Heure_Restant;

	(*Gestion des lectures consignes du mode*)
	Out_Debit_Souf 			:= LIMIT(Cons_Min_Bas_Deb_Ext, Cons_Deb_Soufflage, Cons_Max_Bas_Deb_Ext);
	Out_Debit_Ext 			:= LIMIT(Cons_Min_Bas_Deb_Ext, Cons_Deb_Extraction, Cons_Max_Bas_Deb_Ext);
	Out_Temp_Eau 			:= Cons_Temperature_Eau;

	(*Initialisation des actionneurs non utilisés*)
	Cmd_Douche := FALSE;
	Cmd_Lavabo := FALSE;
	Cmd_Douchette := FALSE;
	Cmd_NEP := FALSE;
	Cmd_Vidange_Douche := FALSE;
	Cmd_Vidange_Lavabo := FALSE;
	Cmd_Electrovanne_Douche := FALSE;
	Cmd_Electrovanne_Lavabo := FALSE;
	Cmd_Prise := FALSE;
	Cmd_Verin_WC_GV := FALSE;
	Cmd_Verin_WC_PV := FALSE;
END_IF;
(*************************************Temporisation du décompte du mode*************************************)
TON_Mode11(
	Enable:= (Mode_11 AND ((E_Vanne_Souf_Bas_Deb_Ouv AND E_Vanne_Ext_Bas_Deb_Ouv) OR Comande_Pause)),
	Pause:= Comande_Pause,
	In_Cons_Seconde:= Tempo_Transition_Seconde,
	In_Cons_Minute:= Tempo_Transition_Minute,
	In_Cons_Heure:= Tempo_Transition_Heure);

(***************************************************************Mode 12 : Mode douche avec vidange transition volume d'eau****************************************************************)
Mode_12 := Numero_Mode = 12 AND Enable;
IF(Mode_12  AND NOT Fin_Action)
	THEN
	(*Gestion du texte*)
	IF(E_Vanne_Vidange_Douche_Ouv)
		THEN
		Out_Texte_FR := 'DOUCHE BONDE OUVERTE ET VOLUME';
		Out_Texte_ENG := 'SHOWER WITH DRAIN AND VOLUME';
		ELSE
		Out_Texte_FR := 'DOUCHE BONDE OUVERTE ET VOLUME - OUVERTURE BONDE';
		Out_Texte_ENG :=  'SHOWER WITH DRAIN AND VOLUME - OPENING DRAIN';
	END_IF;

	(*Gestion de la commande de l'électrovanne et de la vidange*)
	Cmd_Vidange_Douche := TRUE;
	IF(E_Vanne_Vidange_Douche_Ouv)
		THEN
		Cmd_Electrovanne_Douche := TRUE;
		ELSE
		Cmd_Electrovanne_Douche := FALSE;
	END_IF;

	(*Gestion de l'offset*)
	Calcul_Offset_Mode12 := (Tab_MES_Sonde_Debit_Alim_Douche.R_MesCor  / 60.0) + Garde_Deau_Douche;

	(*Gestion du volume d'eau dans la cabine*)
	Integr_Vol_Eau_Mode12(Enable:= Cmd_Electrovanne_Douche,
	Mes_Debit_Eau:= Tab_MES_Sonde_Debit_Alim_Douche.R_MesCor );
	IF((Integr_Vol_Eau_Mode12.Volume_Eau)  >= (Cons_Volume_Eau_Douche + Trop_Plein_Douche - Garde_Deau_Douche))
		THEN
		Cmd_Electrovanne_Douche := FALSE;
		R_TRIG_Mode12(CLK := TRUE);
	END_IF;

	(*Gestion des lectures consignes du mode*)
	Out_Volume_Eau_Douche := Integr_Vol_Eau_Mode12.Volume_Eau;
	Out_Volume_Eau_Lavabo := 0.0;
	Out_Debit_Souf := Cons_Deb_Soufflage;
	Out_Debit_Ext := Cons_Deb_Extraction;
	Out_Temp_Eau := Cons_Temperature_Eau;

	(*Initialisation des actionneurs non utilisés*)
	Cmd_Lavabo := FALSE;
	Cmd_Douche := FALSE;
	Cmd_Douchette := FALSE;
	Cmd_NEP := FALSE;
	Cmd_Vidange_Lavabo := FALSE;
	Cmd_Electrovanne_Lavabo := FALSE;
	Cmd_Prise := FALSE;
	Cmd_Verin_WC_GV := FALSE;
	Cmd_Verin_WC_PV := FALSE;
	ELSE
	R_TRIG_Mode12(CLK := FALSE);
	Integr_Vol_Eau_Mode12(Enable:= FALSE,
	Mes_Debit_Eau:= E_Sonde_Debit_Alim_Douche);
END_IF;

(***************************************************************Mode 13 : Mode douche sans vidange transition volume d'eau****************************************************************)
Mode_13 := Numero_Mode = 13 AND Enable;
IF(Mode_13  AND NOT Fin_Action)
	THEN
	(*Gestion du texte*)
	IF(E_Vanne_Vidange_Douche_Ferm)
		THEN
		Out_Texte_FR := 'DOUCHE BONDE FERMEE ET VOLUME';
		Out_Texte_ENG := 'SHOWER WITHOUT DRAIN AND VOLUME';
		ELSE
		Out_Texte_FR := 'DOUCHE BONDE FERMEE ET VOLUME - FERMETURE BONDE';
		Out_Texte_ENG := 'SHOWER WITHOUT DRAIN AND VOLUME - CLOSING DRAIN';
	END_IF;

	(*Gestion de la commande de l'électrovanne*)
	Cmd_Vidange_Douche := FALSE;
	IF(E_Vanne_Vidange_Douche_Ferm)
		THEN
		Cmd_Electrovanne_Douche := TRUE;
		ELSE
		Cmd_Electrovanne_Douche := FALSE;
	END_IF;

	(*Gestion de l'offset*)
	Calcul_Offset_Mode13 := (Tab_MES_Sonde_Debit_Alim_Douche.R_MesCor  / 60.0) + Garde_Deau_Douche;

	(*Gestion du volume d'eau dans la cabine*)
	Integr_Vol_Eau_Mode13(Enable:= Cmd_Electrovanne_Douche,
	Mes_Debit_Eau:= Tab_MES_Sonde_Debit_Alim_Douche.R_MesCor );
	IF((Integr_Vol_Eau_Mode13.Volume_Eau)  >= (Cons_Volume_Eau_Douche + Trop_Plein_Douche - Garde_Deau_Douche))
		THEN
		Cmd_Electrovanne_Douche := FALSE;
		R_TRIG_Mode13(CLK := TRUE);
	END_IF;

	(*Gestion des lectures consignes du mode*)
	Out_Volume_Eau_Douche := Integr_Vol_Eau_Mode13.Volume_Eau;
	Out_Volume_Eau_Lavabo := 0.0;
	Out_Debit_Souf := Cons_Deb_Soufflage;
	Out_Debit_Ext := Cons_Deb_Extraction;
	Out_Temp_Eau := Cons_Temperature_Eau;

	(*Initialisation des actionneurs non utilisés*)
	Cmd_Lavabo := FALSE;
	Cmd_Douche := FALSE;
	Cmd_Douchette := FALSE;
	Cmd_NEP := FALSE;
	Cmd_Vidange_Lavabo := FALSE;
	Cmd_Electrovanne_Lavabo := FALSE;
	Cmd_Prise := FALSE;
	Cmd_Verin_WC_GV := FALSE;
	Cmd_Verin_WC_PV := FALSE;
	ELSE
	R_TRIG_Mode13(CLK := FALSE);
	Integr_Vol_Eau_Mode13(Enable:= FALSE,
	Mes_Debit_Eau:= E_Sonde_Debit_Alim_Douche);
END_IF;

(***************************************************************Mode 14 : Mode lavabo avec vidange transition volume d'eau****************************************************************)
Mode_14 := Numero_Mode = 14 AND Enable;
IF(Mode_14  AND NOT Fin_Action)
	THEN
	(*Gestion du texte*)
	IF(E_Vanne_Vidange_Lavabo_Ouv)
		THEN
		Out_Texte_FR := 'LAVABO BONDE OUVERTE ET VOLUME';
		Out_Texte_ENG := 'SINK WITH DRAIN ET VOLUME';
		ELSE
		Out_Texte_FR := 'LAVABO BONDE OUVERTE ET VOLUME - OUVERTURE BONDE';
		Out_Texte_ENG := 'SINK WITH DRAIN AND VOLUME - OPENING DRAIN';
	END_IF;

	(*Gestion de la commande de l'électrovanne et de la vidange*)
	Cmd_Vidange_Lavabo := TRUE;
	IF(E_Vanne_Vidange_Lavabo_Ouv)
		THEN
		Cmd_Electrovanne_Lavabo := TRUE;
		ELSE
		Cmd_Electrovanne_Lavabo := FALSE;
	END_IF;

	(*Gestion de l'offset*)
	Calcul_Offset_Mode14 := (Tab_MES_Sonde_Debit_Alim_Lavabo.R_MesCor  / 60.0) + Garde_Deau_Lavabo;

	(*Gestion du volume d'eau dans la cabine*)
	Integr_Vol_Eau_Mode14(Enable:= Cmd_Electrovanne_Lavabo,
	Mes_Debit_Eau := Tab_MES_Sonde_Debit_Alim_Lavabo.R_MesCor );
	IF((Integr_Vol_Eau_Mode14.Volume_Eau)  >= (Cons_Volume_Eau_Lavabo + Trop_Plein_Lavabo - Garde_Deau_Lavabo))
		THEN
		Cmd_Electrovanne_Lavabo := FALSE;
		R_TRIG_Mode14(CLK := TRUE);
	END_IF;

	(*Gestion des lectures consignes du mode*)
	Out_Volume_Eau_Douche := 0.0;
	Out_Volume_Eau_Lavabo := Integr_Vol_Eau_Mode14.Volume_Eau;
	Out_Debit_Souf := Cons_Deb_Soufflage;
	Out_Debit_Ext := Cons_Deb_Extraction;
	Out_Temp_Eau := Cons_Temperature_Eau;

	(*Initialisation des actionneurs non utilisés*)
	Cmd_Lavabo := FALSE;
	Cmd_Douche := FALSE;
	Cmd_Douchette := FALSE;
	Cmd_NEP := FALSE;
	Cmd_Vidange_Douche := FALSE;
	Cmd_Electrovanne_Douche := FALSE;
	Cmd_Prise := FALSE;
	Cmd_Verin_WC_GV := FALSE;
	Cmd_Verin_WC_PV := FALSE;
	ELSE
	R_TRIG_Mode14(CLK := FALSE);
	Integr_Vol_Eau_Mode14(Enable:= FALSE,
	Mes_Debit_Eau := E_Sonde_Debit_Alim_Lavabo);
END_IF;

(***************************************************************Mode 15 : Mode lavabo sans vidange transition volume d'eau****************************************************************)
Mode_15 := Numero_Mode = 15 AND Enable;
IF(Mode_15  AND NOT Fin_Action)
	THEN
	(*Gestion du texte*)
	IF(E_Vanne_Vidange_Lavabo_Ferm)
		THEN
		Out_Texte_FR := 'LAVABO BONDE FERMEE ET VOLUME';
		Out_Texte_ENG := 'SINK WITHOUT DRAIN AND VOLUME';
		ELSE
		Out_Texte_FR := 'LAVABO BONDE FERMEE ET VOLUME - FERMETURE BONDE';
		Out_Texte_ENG := 'SINK WITHOUT DRAIN AND VOLUME - CLOSING DRAIN';
	END_IF;

	(*Gestion de la commande de l'électrovanne*)
	Cmd_Vidange_Lavabo := FALSE;
	IF(E_Vanne_Vidange_Lavabo_Ferm)
		THEN
		Cmd_Electrovanne_Lavabo := TRUE;
		ELSE
		Cmd_Electrovanne_Lavabo := FALSE;
	END_IF;

	(*Gestion de l'offset*)
	Calcul_Offset_Mode15 := (Tab_MES_Sonde_Debit_Alim_Lavabo.R_MesCor  / 60.0) + Garde_Deau_Lavabo;

	(*Gestion du volume d'eau dans la cabine*)
	Integr_Vol_Eau_Mode15(Enable:= Cmd_Electrovanne_Lavabo,
	Mes_Debit_Eau:= Tab_MES_Sonde_Debit_Alim_Lavabo.R_MesCor );
	IF((Integr_Vol_Eau_Mode15.Volume_Eau)  >= (Cons_Volume_Eau_Lavabo + Trop_Plein_Lavabo - Garde_Deau_Lavabo))
		THEN
		Cmd_Electrovanne_Lavabo := FALSE;
		R_TRIG_Mode15(CLK := TRUE);
	END_IF;

	(*Gestion des lectures consignes du mode*)
	Out_Volume_Eau_Douche := 0.0;
	Out_Volume_Eau_Lavabo := Integr_Vol_Eau_Mode15.Volume_Eau;
	Out_Debit_Souf := Cons_Deb_Soufflage;
	Out_Debit_Ext := Cons_Deb_Extraction;
	Out_Temp_Eau := Cons_Temperature_Eau;

	(*Initialisation des actionneurs non utilisés*)
	Cmd_Lavabo := FALSE;
	Cmd_Douche := FALSE;
	Cmd_Douchette := FALSE;
	Cmd_NEP := FALSE;
	Cmd_Vidange_Douche := FALSE;
	Cmd_Electrovanne_Douche := FALSE;
	Cmd_Prise := FALSE;
	Cmd_Verin_WC_GV := FALSE;
	Cmd_Verin_WC_PV := FALSE;
	ELSE
	R_TRIG_Mode15(CLK := FALSE);
	Integr_Vol_Eau_Mode15(Enable:= FALSE,
	Mes_Debit_Eau:= E_Sonde_Debit_Alim_Lavabo);
END_IF;

(****************************************************************Mode 16 : Mode Douche avec vidange transition BP****************************************************************)
Mode_16 := Numero_Mode = 16 AND Enable;
(*Validation de l'étape suivante*)
F_TRIG_Texte16(CLK:= (Valid_Texte AND Mode_16));
IF(Mode_16 AND NOT Fin_Action)
	THEN
	(*Gestion du texte*)
	IF(E_Vanne_Vidange_Douche_Ouv)
		THEN
		Out_Texte_FR := 'DOUCHE BONDE OUVERTE ET BOUTON';
		Out_Texte_ENG := 'SHOWER WITH DRAIN WITH BUTTON';
		ELSE
		Out_Texte_FR := 'DOUCHE BONDE OUVERTE ET BOUTON - OUVERTURE BONDE';
		Out_Texte_ENG := 'SHOWER WITH DRAIN WITH BUTTON - OPENING DRAIN';
	END_IF;

	(*Gestion de la commande de la douche avec vidange douche*)
	Cmd_Vidange_Douche := TRUE;
	IF(E_Vanne_Vidange_Douche_Ouv)
		THEN
		Cmd_Douche := TRUE;
		IF(Option_Debitmetre_Douche)
			THEN
				Cmd_Electrovanne_Douche := TRUE;
			ELSE
				Cmd_Electrovanne_Douche := FALSE;
		END_IF;
		ELSE
		Cmd_Douche := FALSE;
		Cmd_Electrovanne_Douche := FALSE;
	END_IF;

	IF(Comande_Pause)
		THEN
		Cmd_Douche := FALSE;
		Cmd_Electrovanne_Douche := FALSE;
	END_IF;

	(*Gestion des lectures consignes du mode*)
	Out_Debit_Souf 			:= Cons_Deb_Soufflage;
	Out_Debit_Ext 			:= Cons_Deb_Extraction;
	Out_Temp_Eau 			:= Cons_Temperature_Eau;

	(*Initialisation des actionneurs non utilisés*)
	Cmd_Lavabo := FALSE;
	Cmd_Douchette := FALSE;
	Cmd_NEP := FALSE;
	Cmd_Vidange_Lavabo := FALSE;
	Cmd_Electrovanne_Lavabo := FALSE;
	Cmd_Prise := FALSE;
	Cmd_Verin_WC_GV := FALSE;
	Cmd_Verin_WC_PV := FALSE;
END_IF;

(****************************************************************Mode 17 : Mode Lavabo avec vidange transition BP****************************************************************)
Mode_17 := Numero_Mode = 17 AND Enable;
(*Validation de l'étape suivante*)
F_TRIG_Texte17(CLK:= (Valid_Texte AND Mode_17));
IF(Mode_17 AND NOT Fin_Action)
	THEN
	(*Gestion du texte*)
	IF(E_Vanne_Vidange_Lavabo_Ouv)
		THEN
		Out_Texte_FR := 'DOUCHE BONDE OUVERTE ET BOUTON';
		Out_Texte_ENG := 'SINK WITH DRAIN WITH BUTTON';
		ELSE
		Out_Texte_FR := 'DOUCHE BONDE OUVERTE ET BOUTON - OUVERTURE BONDE';
		Out_Texte_ENG := 'SINK WITH DRAIN WITH BUTTON - OPENING DRAIN';
	END_IF;

	(*Gestion de la commande du lavabo avec vidange lavabo*)
	Cmd_Vidange_Lavabo := TRUE;
	IF(E_Vanne_Vidange_Lavabo_Ouv)
		THEN
		Cmd_Lavabo := TRUE;
		IF(Option_Debitmetre_Lavabo)
			THEN
				Cmd_Electrovanne_Lavabo := TRUE;
			ELSE
				Cmd_Electrovanne_Lavabo := FALSE;
		END_IF;
		ELSE
		Cmd_Lavabo := FALSE;
		Cmd_Electrovanne_Lavabo := FALSE;
	END_IF;

	IF(Comande_Pause)
		THEN
		Cmd_Lavabo := FALSE;
		Cmd_Electrovanne_Lavabo := FALSE;
	END_IF;

	(*Gestion des lectures consignes du mode*)
	Out_Debit_Souf 			:= Cons_Deb_Soufflage;
	Out_Debit_Ext 			:= Cons_Deb_Extraction;
	Out_Temp_Eau 			:= Cons_Temperature_Eau;

	(*Initialisation des actionneurs non utilisés*)
	Cmd_Douche := FALSE;
	Cmd_Douchette := FALSE;
	Cmd_NEP := FALSE;
	Cmd_Vidange_Douche := FALSE;
	Cmd_Electrovanne_Douche := FALSE;
	Cmd_Prise := FALSE;
	Cmd_Verin_WC_GV := FALSE;
	Cmd_Verin_WC_PV := FALSE;
END_IF;

(****************************************************************Mode 18 : Mode lavage NEP eau chaude****************************************************************)
Mode_18 := Numero_Mode = 18 AND Enable;
IF(Mode_18  AND NOT Fin_Action)
	THEN
	(*Gestion du texte*)
	IF(E_Vanne_Vidange_Douche_Ouv)
		THEN
		Out_Texte_FR := 'LAVAGE EAU CHAUDE';
		Out_Texte_ENG := 'HOT WATER CLEANING';
		ELSE
		Out_Texte_FR := 'LAVAGE EAU CHAUDE - OUVERTURE BONDE';
		Out_Texte_ENG :=  'HOT WATER CLEANING - OPENING DRAIN';
	END_IF;
	IF(RS_Fin_Mode_18.Q1)
		THEN
		Out_Texte_FR := 'LAVAGE EAU CHAUDE - ARRET LAVAGE';
		Out_Texte_ENG := 'HOT WATER CLEANING - STOPING CLEANING';
	END_IF;

	(*Gestion de la commande de la NEP et de la vidange*)
	Cmd_Vidange_Douche := TRUE;
	(*Ouverture à 100% de la vanne 3 voies pour le mode chaud*)
	Out_Cons_V3V_Eau_Mitig := 100.0;
	IF( RS_Fin_Mode_18.Q1)
		THEN
		Out_Restant_Seconde := 0.0;
		Out_Restant_Minute := 0.0;
		Out_Restant_Heure := 0.0;
		Cmd_NEP := FALSE;
		ELSE
		IF(E_Vanne_Vidange_Douche_Ouv)
			THEN
			Cmd_NEP := TRUE;
			ELSE
			Cmd_NEP := FALSE;
		END_IF;
	END_IF;

	(*Gestion de la commande pause*)
	IF(Comande_Pause)
		THEN
		Cmd_NEP := FALSE;
	END_IF;

	(*Gestion du décompte de la temporisation du mode*)
	Out_Restant_Seconde := TON_Mode18.Seconde_Restant;
	Out_Restant_Minute := TON_Mode18.Minute_Restant;
	Out_Restant_Heure := TON_Mode18.Heure_Restant;

	(*Gestion des lectures consignes du mode*)
	Out_Debit_Souf 			:= Cons_Deb_Soufflage;
	Out_Debit_Ext 			:= Cons_Deb_Extraction;
	Out_Temp_Eau 			:= Cons_Temperature_Eau;

	(*Initialisation des actionneurs non utilisés*)
	Cmd_Douche := FALSE;
	Cmd_Lavabo := FALSE;
	Cmd_Douchette := FALSE;
	Cmd_Vidange_Lavabo := FALSE;
	Cmd_Electrovanne_Douche := FALSE;
	Cmd_Electrovanne_Lavabo := FALSE;
	Cmd_Prise := FALSE;
	Cmd_Verin_WC_GV := FALSE;
	Cmd_Verin_WC_PV := FALSE;
END_IF;
(*************************************Temporisation du décompte du mode*************************************)
TON_Mode18(
Enable:= (Mode_18 AND ((E_Vanne_Vidange_Douche_Ouv AND E_Vanne_Alim_NEP_Ouv) OR Comande_Pause)),
Pause:= Comande_Pause,
In_Cons_Seconde:= Tempo_Transition_Seconde,
In_Cons_Minute:= Tempo_Transition_Minute,
In_Cons_Heure:= Tempo_Transition_Heure);

(*Activation de la fin du mode*)
RS_Fin_Mode_18(SET:= TON_Mode18.Q, RESET1:= NOT Mode_18);
IF( RS_Fin_Mode_18.Q1)
	THEN
	Out_Restant_Seconde := 0.0;
	Out_Restant_Minute := 0.0;
	Out_Restant_Heure := 0.0;
END_IF;

(****************************************************************Mode 19 : Mode lavage NEP eau froide****************************************************************)
Mode_19 := Numero_Mode = 19 AND Enable;
IF(Mode_19  AND NOT Fin_Action)
	THEN
	(*Gestion du texte*)
	IF(E_Vanne_Vidange_Douche_Ouv)
		THEN
		Out_Texte_FR := 'LAVAGE EAU FROIDE';
		Out_Texte_ENG := 'COLD WATER CLEANING';
		ELSE
		Out_Texte_FR := 'LAVAGE EAU FROIDE - OUVERTURE BONDE';
		Out_Texte_ENG :=  'COLD WATER CLEANING - OPENING DRAIN';
	END_IF;
	IF(RS_Fin_Mode_19.Q1)
		THEN
		Out_Texte_FR := 'LAVAGE EAU FROIDE - ARRET LAVAGE';
		Out_Texte_ENG := 'COLD WATER CLEANING - STOPING CLEANING';
	END_IF;

	(*Gestion de la commande de la NEP et de la vidange*)
	Cmd_Vidange_Douche := TRUE;
	(*Ouverture à 0% de la vanne 3 voies pour le mode froid*)
	Out_Cons_V3V_Eau_Mitig := 0.0;
	IF( RS_Fin_Mode_19.Q1)
		THEN
		Out_Restant_Seconde := 0.0;
		Out_Restant_Minute := 0.0;
		Out_Restant_Heure := 0.0;
		Cmd_NEP := FALSE;
		ELSE
		IF(E_Vanne_Vidange_Douche_Ouv)
			THEN
			Cmd_NEP := TRUE;
			ELSE
			Cmd_NEP := FALSE;
		END_IF;
	END_IF;

	(*Gestion de la commande pause*)
	IF(Comande_Pause)
		THEN
		Cmd_NEP := FALSE;
	END_IF;

	(*Gestion du décompte de la temporisation du mode*)
	Out_Restant_Seconde := TON_Mode19.Seconde_Restant;
	Out_Restant_Minute := TON_Mode19.Minute_Restant;
	Out_Restant_Heure := TON_Mode19.Heure_Restant;

	(*Gestion des lectures consignes du mode*)
	Out_Debit_Souf 			:= Cons_Deb_Soufflage;
	Out_Debit_Ext 			:= Cons_Deb_Extraction;
	Out_Temp_Eau 			:= Cons_Temperature_Eau;

	(*Initialisation des actionneurs non utilisés*)
	Cmd_Douche := FALSE;
	Cmd_Lavabo := FALSE;
	Cmd_Douchette := FALSE;
	Cmd_Vidange_Lavabo := FALSE;
	Cmd_Electrovanne_Douche := FALSE;
	Cmd_Electrovanne_Lavabo := FALSE;
	Cmd_Prise := FALSE;
	Cmd_Verin_WC_GV := FALSE;
	Cmd_Verin_WC_PV := FALSE;
END_IF;
(*************************************Temporisation du décompte du mode*************************************)
TON_Mode19(
Enable:= (Mode_19 AND ((E_Vanne_Vidange_Douche_Ouv AND E_Vanne_Alim_NEP_Ouv) OR Comande_Pause)),
Pause:= Comande_Pause,
In_Cons_Seconde:= Tempo_Transition_Seconde,
In_Cons_Minute:= Tempo_Transition_Minute,
In_Cons_Heure:= Tempo_Transition_Heure);

(*Activation de la fin du mode*)
RS_Fin_Mode_19(SET:= TON_Mode19.Q, RESET1:= NOT Mode_19);
IF( RS_Fin_Mode_19.Q1)
	THEN
	Out_Restant_Seconde := 0.0;
	Out_Restant_Minute := 0.0;
	Out_Restant_Heure := 0.0;
END_IF;

